KUKA KRL program: f1_Kuka_APT232T02S32.SRC

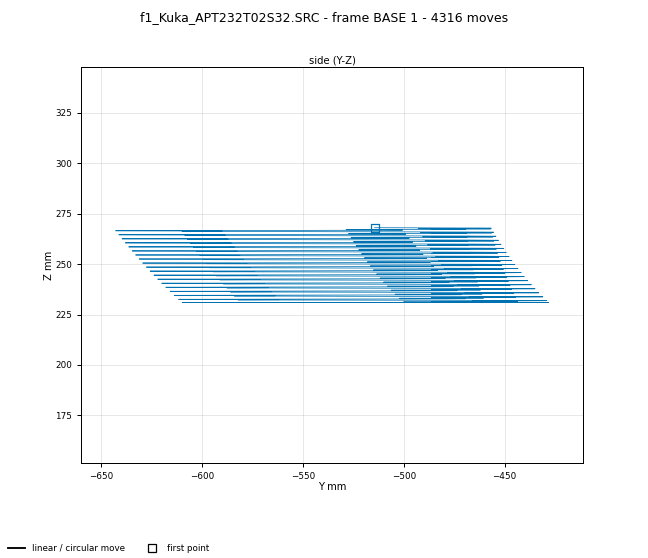
[picture p0: tool path of f1_Kuka_APT232T02S32.SRC in frame BASE 1, 4316 of 4317 moves have a stored position in this frame; points joined in program order, loops and branches not executed]
&ACCESS RVP
&REL 2
&PARAM TEMPLATE = C:\KRC\Roboter\Template\vorgabe
&PARAM EDITMASK = *
DEF f1_Kuka_APT232T02S32()


;FOLD INI;%{PE}%V3.2.0,%MKUKATPBASIS,%CINIT,%VCOMMON,%P
  ;FOLD BAS INI;%{E}%V3.2.0,%MKUKATPBASIS,%CINIT,%VINIT,%P
    GLOBAL INTERRUPT DECL 3 WHEN $STOPMESS==TRUE DO IR_STOPM ( )
    INTERRUPT ON 3
    BAS (#INITMOV,0 )
  ;ENDFOLD (BAS INI)
  ;FOLD USER INI;%{E}%V3.2.0,%MKUKATPUSER,%CINIT,%VINIT,%P
    ;Make your modifications here
  ;ENDFOLD (USER INI)
;ENDFOLD (INI)


;*** Make Null PTP Move
  PTP $pos_act

;*** Auto Load The Correct TOOL Data
  $tool=tool_data[2]

;*** Auto Load The Correct BASE Data
  $base=base_data[1]

  $ADVANCE = 5

;*** Restate Last Velocity
MMPM(30000.0)
SetRPM(8000)
LIN {X -0.230,Y -514.426,Z 267.989,A 0.000,B 0.000,C 90.000,E1 213.992} C_DIS
LIN {X 0.196,Y -508.743,Z 267.977,A 0.000,B 0.000,C 90.000,E1 211.878} C_DIS
LIN {X 0.196,Y -503.250,Z 267.966,A 0.000,B 0.000,C 90.000,E1 209.795} C_DIS
LIN {X -0.056,Y -498.886,Z 267.956,A 0.000,B 0.000,C 90.000,E1 208.025} C_DIS
LIN {X 0.152,Y -492.690,Z 267.941,A 0.000,B 0.000,C 90.000,E1 205.283} C_DIS
LIN {X 0.150,Y -488.290,Z 267.929,A 0.000,B 0.000,C 90.000,E1 203.153} C_DIS
LIN {X -0.154,Y -484.154,Z 267.917,A 0.000,B 0.000,C 90.000,E1 201.046} C_DIS
LIN {X 0.157,Y -479.821,Z 267.903,A 0.000,B 0.000,C 90.000,E1 198.544} C_DIS
LIN {X 0.025,Y -475.933,Z 267.889,A 0.000,B 0.000,C 90.000,E1 196.079} C_DIS
LIN {X 0.194,Y -471.593,Z 267.872,A 0.000,B 0.000,C 90.000,E1 192.939} C_DIS
LIN {X -0.221,Y -469.656,Z 267.863,A 0.000,B 0.000,C 90.000,E1 191.422} C_DIS
LIN {X 0.157,Y -466.683,Z 267.849,A 0.000,B 0.000,C 90.000,E1 188.859} C_DIS
LIN {X -0.167,Y -464.095,Z 267.835,A 0.000,B 0.000,C 90.000,E1 186.372} C_DIS
LIN {X 0.063,Y -462.670,Z 267.827,A 0.000,B 0.000,C 90.000,E1 184.759} C_DIS
LIN {X 0.115,Y -460.444,Z 267.811,A 0.000,B 0.000,C 90.000,E1 181.892} C_DIS
LIN {X 0.087,Y -458.680,Z 267.795,A 0.000,B 0.000,C 90.000,E1 179.026} C_DIS
LIN {X 0.013,Y -457.404,Z 267.779,A 0.000,B 0.000,C 90.000,E1 176.159} C_DIS
LIN {X 0.059,Y -456.833,Z 267.766,A 0.000,B 0.000,C 90.000,E1 173.913} C_DIS
LIN {X -0.071,Y -456.684,Z 267.756,A 0.000,B 0.000,C 90.000,E1 172.008} C_DIS
LIN {X -0.145,Y -456.659,Z 267.741,A 0.000,B 0.000,C 90.000,E1 169.454} C_DIS
LIN {X 0.170,Y -457.094,Z 267.729,A 0.000,B 0.000,C 90.000,E1 167.173} C_DIS
LIN {X 0.039,Y -457.494,Z 267.720,A 0.000,B 0.000,C 90.000,E1 165.589} C_DIS
LIN {X 0.182,Y -459.071,Z 267.700,A 0.000,B 0.000,C 90.000,E1 162.054} C_DIS
LIN {X -0.015,Y -461.188,Z 267.685,A 0.000,B 0.000,C 90.000,E1 159.209} C_DIS
LIN {X 0.063,Y -463.174,Z 267.672,A 0.000,B 0.000,C 90.000,E1 156.975} C_DIS
LIN {X -0.031,Y -466.661,Z 267.655,A 0.000,B 0.000,C 90.000,E1 153.819} C_DIS
LIN {X -0.099,Y -470.005,Z 267.641,A 0.000,B 0.000,C 90.000,E1 151.307} C_DIS
LIN {X 0.204,Y -473.267,Z 267.628,A 0.000,B 0.000,C 90.000,E1 149.076} C_DIS
LIN {X -0.166,Y -476.278,Z 267.618,A 0.000,B 0.000,C 90.000,E1 147.248} C_DIS
LIN {X -0.209,Y -479.468,Z 267.608,A 0.000,B 0.000,C 90.000,E1 145.388} C_DIS
LIN {X 0.091,Y -482.592,Z 267.597,A 0.000,B 0.000,C 90.000,E1 143.497} C_DIS
LIN {X -0.019,Y -485.558,Z 267.587,A 0.000,B 0.000,C 90.000,E1 141.662} C_DIS
LIN {X -0.030,Y -487.431,Z 267.580,A 0.000,B 0.000,C 90.000,E1 140.436} C_DIS
LIN {X -0.247,Y -489.510,Z 267.572,A 0.000,B 0.000,C 90.000,E1 138.933} C_DIS
LIN {X 0.062,Y -490.896,Z 267.565,A 0.000,B 0.000,C 90.000,E1 137.676} C_DIS
LIN {X -0.107,Y -491.742,Z 267.560,A 0.000,B 0.000,C 90.000,E1 136.782} C_DIS
LIN {X -0.293,Y -492.387,Z 267.555,A 0.000,B 0.000,C 90.000,E1 135.891} C_DIS
LIN {X 0.054,Y -492.760,Z 267.548,A 0.000,B 0.000,C 90.000,E1 134.636} C_DIS
LIN {X 0.233,Y -492.889,Z 267.543,A 0.000,B 0.000,C 90.000,E1 133.704} C_DIS
LIN {X -0.277,Y -492.766,Z 267.538,A 0.000,B 0.000,C 90.000,E1 132.852} C_DIS
LIN {X -0.090,Y -492.444,Z 267.533,A 0.000,B 0.000,C 90.000,E1 131.919} C_DIS
LIN {X -0.067,Y -491.559,Z 267.526,A 0.000,B 0.000,C 90.000,E1 130.701} C_DIS
LIN {X -0.061,Y -490.329,Z 267.519,A 0.000,B 0.000,C 90.000,E1 129.483} C_DIS
LIN {X -0.006,Y -488.945,Z 267.513,A 0.000,B 0.000,C 90.000,E1 128.257} C_DIS
LIN {X 0.033,Y -487.284,Z 267.506,A 0.000,B 0.000,C 90.000,E1 127.030} C_DIS
LIN {X 0.045,Y -485.471,Z 267.499,A 0.000,B 0.000,C 90.000,E1 125.804} C_DIS
LIN {X -0.039,Y -482.830,Z 267.490,A 0.000,B 0.000,C 90.000,E1 124.278} C_DIS
LIN {X -0.173,Y -480.059,Z 267.482,A 0.000,B 0.000,C 90.000,E1 122.752} C_DIS
LIN {X 0.034,Y -477.274,Z 267.473,A 0.000,B 0.000,C 90.000,E1 121.180} C_DIS
LIN {X 0.103,Y -474.436,Z 267.465,A 0.000,B 0.000,C 90.000,E1 119.617} C_DIS
LIN {X -0.166,Y -470.393,Z 267.453,A 0.000,B 0.000,C 90.000,E1 117.462} C_DIS
LIN {X 0.196,Y -467.495,Z 267.444,A 0.000,B 0.000,C 90.000,E1 115.848} C_DIS
LIN {X 0.156,Y -463.423,Z 267.432,A 0.000,B 0.000,C 90.000,E1 113.643} C_DIS
LIN {X 0.053,Y -461.128,Z 267.424,A 0.000,B 0.000,C 90.000,E1 112.386} C_DIS
LIN {X 0.164,Y -458.908,Z 267.417,A 0.000,B 0.000,C 90.000,E1 111.099} C_DIS
LIN {X -0.015,Y -456.909,Z 267.411,A 0.000,B 0.000,C 90.000,E1 109.939} C_DIS
LIN {X -0.055,Y -456.917,Z 267.411,A 0.000,B 0.000,C 90.000,E1 109.939} C_DIS
LIN {X 0.148,Y -457.785,Z 267.409,A 0.000,B 0.000,C 90.000,E1 109.504} C_DIS
LIN {X 0.113,Y -466.564,Z 267.386,A 0.000,B 0.000,C 90.000,E1 105.371} C_DIS
LIN {X 0.036,Y -467.351,Z 267.384,A 0.000,B 0.000,C 90.000,E1 105.064} C_DIS
LIN {X -0.160,Y -468.007,Z 267.382,A 0.000,B 0.000,C 90.000,E1 104.773} C_DIS
LIN {X -0.198,Y -476.222,Z 267.356,A 0.000,B 0.000,C 90.000,E1 100.074} C_DIS
LIN {X 0.056,Y -482.120,Z 267.330,A 0.000,B 0.000,C 90.000,E1 95.391} C_DIS
LIN {X -0.195,Y -485.524,Z 267.304,A 0.000,B 0.000,C 90.000,E1 90.802} C_DIS
LIN {X -0.161,Y -486.381,Z 267.281,A 0.000,B 0.000,C 90.000,E1 86.502} C_DIS
LIN {X 0.148,Y -486.354,Z 267.279,A 0.000,B 0.000,C 90.000,E1 86.159} C_DIS
LIN {X 0.227,Y -484.671,Z 267.253,A 0.000,B 0.000,C 90.000,E1 81.546} C_DIS
LIN {X 0.116,Y -480.589,Z 267.228,A 0.000,B 0.000,C 90.000,E1 76.937} C_DIS
LIN {X -0.172,Y -479.679,Z 267.224,A 0.000,B 0.000,C 90.000,E1 76.353} C_DIS
LIN {X -0.137,Y -474.020,Z 267.200,A 0.000,B 0.000,C 90.000,E1 72.000} C_DIS
LIN {X 0.177,Y -469.391,Z 267.186,A 0.000,B 0.000,C 90.000,E1 69.518} C_DIS
LIN {X 0.138,Y -469.387,Z 267.186,A 0.000,B 0.000,C 90.000,E1 69.518} C_DIS
LIN {X -0.086,Y -473.477,Z 267.177,A 0.000,B 0.000,C 90.000,E1 67.922} C_DIS
LIN {X -0.070,Y -478.382,Z 267.167,A 0.000,B 0.000,C 90.000,E1 66.049} C_DIS
LIN {X 0.060,Y -482.474,Z 267.158,A 0.000,B 0.000,C 90.000,E1 64.485} C_DIS
LIN {X -0.171,Y -487.487,Z 267.148,A 0.000,B 0.000,C 90.000,E1 62.666} C_DIS
LIN {X -0.098,Y -491.783,Z 267.140,A 0.000,B 0.000,C 90.000,E1 61.129} C_DIS
LIN {X 0.124,Y -496.998,Z 267.129,A 0.000,B 0.000,C 90.000,E1 59.282} C_DIS
LIN {X 0.139,Y -500.549,Z 267.123,A 0.000,B 0.000,C 90.000,E1 58.074} C_DIS
LIN {X -0.219,Y -504.000,Z 267.116,A 0.000,B 0.000,C 90.000,E1 56.914} C_DIS
LIN {X 0.173,Y -507.369,Z 267.109,A 0.000,B 0.000,C 90.000,E1 55.674} C_DIS
LIN {X 0.110,Y -511.278,Z 267.101,A 0.000,B 0.000,C 90.000,E1 54.196} C_DIS
LIN {X -0.219,Y -514.259,Z 267.095,A 0.000,B 0.000,C 90.000,E1 53.050} C_DIS
LIN {X 0.217,Y -516.997,Z 267.088,A 0.000,B 0.000,C 90.000,E1 51.823} C_DIS
LIN {X 0.231,Y -520.051,Z 267.080,A 0.000,B 0.000,C 90.000,E1 50.356} C_DIS
LIN {X -0.051,Y -522.220,Z 267.073,A 0.000,B 0.000,C 90.000,E1 49.218} C_DIS
LIN {X 0.137,Y -523.619,Z 267.069,A 0.000,B 0.000,C 90.000,E1 48.324} C_DIS
LIN {X -0.053,Y -524.883,Z 267.064,A 0.000,B 0.000,C 90.000,E1 47.472} C_DIS
LIN {X 0.081,Y -526.244,Z 267.057,A 0.000,B 0.000,C 90.000,E1 46.296} C_DIS
LIN {X -0.145,Y -527.243,Z 267.051,A 0.000,B 0.000,C 90.000,E1 45.162} C_DIS
LIN {X 0.068,Y -527.840,Z 267.046,A 0.000,B 0.000,C 90.000,E1 44.271} C_DIS
LIN {X -0.139,Y -528.298,Z 267.040,A 0.000,B 0.000,C 90.000,E1 43.137} C_DIS
LIN {X 0.039,Y -528.525,Z 267.033,A 0.000,B 0.000,C 90.000,E1 41.962} C_DIS
LIN {X 0.295,Y -528.546,Z 267.028,A 0.000,B 0.000,C 90.000,E1 41.067} C_DIS
LIN {X -0.189,Y -528.403,Z 267.024,A 0.000,B 0.000,C 90.000,E1 40.253} C_DIS
LIN {X 0.074,Y -528.098,Z 267.019,A 0.000,B 0.000,C 90.000,E1 39.358} C_DIS
LIN {X -0.137,Y -527.300,Z 267.011,A 0.000,B 0.000,C 90.000,E1 37.935} C_DIS
LIN {X -0.248,Y -526.425,Z 267.004,A 0.000,B 0.000,C 90.000,E1 36.790} C_DIS
LIN {X 0.057,Y -525.340,Z 266.998,A 0.000,B 0.000,C 90.000,E1 35.598} C_DIS
LIN {X 0.306,Y -523.688,Z 266.990,A 0.000,B 0.000,C 90.000,E1 34.119} C_DIS
LIN {X 0.273,Y -522.280,Z 266.983,A 0.000,B 0.000,C 90.000,E1 32.959} C_DIS
LIN {X -0.110,Y -520.461,Z 266.975,A 0.000,B 0.000,C 90.000,E1 31.544} C_DIS
LIN {X -0.154,Y -518.224,Z 266.965,A 0.000,B 0.000,C 90.000,E1 29.795} C_DIS
LIN {X -0.063,Y -516.128,Z 266.956,A 0.000,B 0.000,C 90.000,E1 28.025} C_DIS
LIN {X 0.197,Y -514.018,Z 266.946,A 0.000,B 0.000,C 90.000,E1 26.232} C_DIS
LIN {X -0.158,Y -511.788,Z 266.934,A 0.000,B 0.000,C 90.000,E1 24.207} C_DIS
LIN {X -0.058,Y -510.297,Z 266.926,A 0.000,B 0.000,C 90.000,E1 22.717} C_DIS
LIN {X 0.224,Y -508.272,Z 266.915,A 0.000,B 0.000,C 90.000,E1 20.610} C_DIS
LIN {X -0.004,Y -506.763,Z 266.905,A 0.000,B 0.000,C 90.000,E1 18.852} C_DIS
LIN {X 0.151,Y -505.095,Z 266.893,A 0.000,B 0.000,C 90.000,E1 16.749} C_DIS
LIN {X 0.183,Y -503.375,Z 266.880,A 0.000,B 0.000,C 90.000,E1 14.356} C_DIS
LIN {X 0.143,Y -501.822,Z 266.863,A 0.000,B 0.000,C 90.000,E1 11.366} C_DIS
LIN {X 0.017,Y -500.880,Z 266.848,A 0.000,B 0.000,C 90.000,E1 8.681} C_DIS
LIN {X -0.219,Y -500.607,Z 266.837,A 0.000,B 0.000,C 90.000,E1 6.606} C_DIS
LIN {X -0.176,Y -500.591,Z 266.822,A 0.000,B 0.000,C 90.000,E1 3.898} C_DIS
LIN {X -0.121,Y -501.117,Z 266.808,A 0.000,B 0.000,C 90.000,E1 1.489} C_DIS
LIN {X -0.044,Y -502.113,Z 266.796,A 0.000,B 0.000,C 90.000,E1 359.198} C_DIS
LIN {X 0.076,Y -503.746,Z 266.782,A 0.000,B 0.000,C 90.000,E1 356.788} C_DIS
LIN {X -0.150,Y -505.603,Z 266.771,A 0.000,B 0.000,C 90.000,E1 354.723} C_DIS
LIN {X -0.073,Y -507.065,Z 266.762,A 0.000,B 0.000,C 90.000,E1 353.223} C_DIS
LIN {X 0.174,Y -512.463,Z 266.743,A 0.000,B 0.000,C 90.000,E1 349.634} C_DIS
LIN {X 0.075,Y -519.137,Z 266.726,A 0.000,B 0.000,C 90.000,E1 346.700} C_DIS
LIN {X 0.181,Y -523.006,Z 266.718,A 0.000,B 0.000,C 90.000,E1 345.227} C_DIS
LIN {X -0.168,Y -526.106,Z 266.712,A 0.000,B 0.000,C 90.000,E1 344.102} C_DIS
LIN {X 0.250,Y -533.219,Z 266.697,A 0.000,B 0.000,C 90.000,E1 341.456} C_DIS
LIN {X 0.138,Y -539.356,Z 266.686,A 0.000,B 0.000,C 90.000,E1 339.464} C_DIS
LIN {X -0.207,Y -546.932,Z 266.673,A 0.000,B 0.000,C 90.000,E1 337.230} C_DIS
LIN {X 0.081,Y -551.791,Z 266.666,A 0.000,B 0.000,C 90.000,E1 335.793} C_DIS
LIN {X -0.049,Y -556.779,Z 266.658,A 0.000,B 0.000,C 90.000,E1 334.409} C_DIS
LIN {X -0.247,Y -563.958,Z 266.647,A 0.000,B 0.000,C 90.000,E1 332.487} C_DIS
LIN {X -0.243,Y -568.105,Z 266.641,A 0.000,B 0.000,C 90.000,E1 331.385} C_DIS
LIN {X -0.073,Y -573.033,Z 266.633,A 0.000,B 0.000,C 90.000,E1 329.999} C_DIS
LIN {X 0.184,Y -577.781,Z 266.626,A 0.000,B 0.000,C 90.000,E1 328.614} C_DIS
LIN {X -0.132,Y -584.424,Z 266.615,A 0.000,B 0.000,C 90.000,E1 326.755} C_DIS
LIN {X 0.003,Y -590.503,Z 266.606,A 0.000,B 0.000,C 90.000,E1 325.135} C_DIS
LIN {X -0.029,Y -596.487,Z 266.598,A 0.000,B 0.000,C 90.000,E1 323.543} C_DIS
LIN {X 0.069,Y -600.158,Z 266.592,A 0.000,B 0.000,C 90.000,E1 322.477} C_DIS
LIN {X -0.010,Y -604.543,Z 266.584,A 0.000,B 0.000,C 90.000,E1 321.170} C_DIS
LIN {X 0.368,Y -608.852,Z 266.577,A 0.000,B 0.000,C 90.000,E1 319.828} C_DIS
LIN {X -0.222,Y -613.909,Z 266.568,A 0.000,B 0.000,C 90.000,E1 318.324} C_DIS
LIN {X 0.267,Y -618.187,Z 266.561,A 0.000,B 0.000,C 90.000,E1 316.986} C_DIS
LIN {X 0.254,Y -620.662,Z 266.557,A 0.000,B 0.000,C 90.000,E1 316.215} C_DIS
LIN {X -0.026,Y -624.392,Z 266.550,A 0.000,B 0.000,C 90.000,E1 314.960} C_DIS
LIN {X -0.116,Y -627.253,Z 266.544,A 0.000,B 0.000,C 90.000,E1 313.947} C_DIS
LIN {X -0.161,Y -629.986,Z 266.538,A 0.000,B 0.000,C 90.000,E1 312.933} C_DIS
LIN {X -0.167,Y -632.434,Z 266.533,A 0.000,B 0.000,C 90.000,E1 311.919} C_DIS
LIN {X -0.147,Y -634.695,Z 266.527,A 0.000,B 0.000,C 90.000,E1 310.906} C_DIS
LIN {X -0.029,Y -636.679,Z 266.522,A 0.000,B 0.000,C 90.000,E1 309.886} C_DIS
LIN {X -0.370,Y -638.383,Z 266.516,A 0.000,B 0.000,C 90.000,E1 308.910} C_DIS
LIN {X 0.206,Y -640.180,Z 266.509,A 0.000,B 0.000,C 90.000,E1 307.604} C_DIS
LIN {X 0.406,Y -641.435,Z 266.503,A 0.000,B 0.000,C 90.000,E1 306.583} C_DIS
LIN {X -0.172,Y -642.058,Z 266.499,A 0.000,B 0.000,C 90.000,E1 305.884} C_DIS
LIN {X 0.157,Y -642.446,Z 266.495,A 0.000,B 0.000,C 90.000,E1 305.105} C_DIS
LIN {X -0.409,Y -642.645,Z 266.491,A 0.000,B 0.000,C 90.000,E1 304.405} C_DIS
LIN {X 0.370,Y -642.696,Z 266.484,A 0.000,B 0.000,C 90.000,E1 303.086} C_DIS
LIN {X 0.339,Y -642.403,Z 266.480,A 0.000,B 0.000,C 90.000,E1 302.339} C_DIS
LIN {X 0.305,Y -641.761,Z 266.476,A 0.000,B 0.000,C 90.000,E1 301.592} C_DIS
LIN {X -0.126,Y -641.196,Z 266.473,A 0.000,B 0.000,C 90.000,E1 301.131} C_DIS
LIN {X -0.175,Y -639.987,Z 266.469,A 0.000,B 0.000,C 90.000,E1 300.384} C_DIS
LIN {X 0.364,Y -638.024,Z 266.463,A 0.000,B 0.000,C 90.000,E1 299.333} C_DIS
LIN {X 0.061,Y -635.155,Z 266.456,A 0.000,B 0.000,C 90.000,E1 298.103} C_DIS
LIN {X -0.324,Y -632.632,Z 266.451,A 0.000,B 0.000,C 90.000,E1 297.129} C_DIS
LIN {X -0.150,Y -629.298,Z 266.444,A 0.000,B 0.000,C 90.000,E1 295.848} C_DIS
LIN {X -0.273,Y -624.517,Z 266.434,A 0.000,B 0.000,C 90.000,E1 294.079} C_DIS
LIN {X 0.067,Y -621.195,Z 266.427,A 0.000,B 0.000,C 90.000,E1 292.770} C_DIS
LIN {X -0.178,Y -615.973,Z 266.415,A 0.000,B 0.000,C 90.000,E1 290.737} C_DIS
LIN {X 0.059,Y -611.666,Z 266.405,A 0.000,B 0.000,C 90.000,E1 288.906} C_DIS
LIN {X -0.044,Y -605.942,Z 266.391,A 0.000,B 0.000,C 90.000,E1 286.315} C_DIS
LIN {X -0.282,Y -601.908,Z 266.379,A 0.000,B 0.000,C 90.000,E1 284.245} C_DIS
LIN {X 0.146,Y -596.652,Z 266.360,A 0.000,B 0.000,C 90.000,E1 280.782} C_DIS
LIN {X -0.261,Y -593.058,Z 266.342,A 0.000,B 0.000,C 90.000,E1 277.644} C_DIS
LIN {X -0.064,Y -590.974,Z 266.326,A 0.000,B 0.000,C 90.000,E1 274.702} C_DIS
LIN {X 0.269,Y -589.995,Z 266.311,A 0.000,B 0.000,C 90.000,E1 272.007} C_DIS
LIN {X 0.003,Y -590.230,Z 266.292,A 0.000,B 0.000,C 90.000,E1 268.568} C_DIS
LIN {X -0.149,Y -592.176,Z 266.273,A 0.000,B 0.000,C 90.000,E1 265.122} C_DIS
LIN {X -0.173,Y -594.805,Z 266.258,A 0.000,B 0.000,C 90.000,E1 262.470} C_DIS
LIN {X -0.052,Y -599.032,Z 266.241,A 0.000,B 0.000,C 90.000,E1 259.285} C_DIS
LIN {X -0.005,Y -601.486,Z 266.232,A 0.000,B 0.000,C 90.000,E1 257.701} C_DIS
LIN {X 0.097,Y -604.047,Z 266.223,A 0.000,B 0.000,C 90.000,E1 256.117} C_DIS
LIN {X -0.192,Y -606.411,Z 266.214,A 0.000,B 0.000,C 90.000,E1 254.574} C_DIS
LIN {X -0.235,Y -607.542,Z 266.210,A 0.000,B 0.000,C 90.000,E1 253.795} C_DIS
LIN {X 0.319,Y -608.398,Z 266.206,A 0.000,B 0.000,C 90.000,E1 252.960} C_DIS
LIN {X 0.298,Y -608.926,Z 266.201,A 0.000,B 0.000,C 90.000,E1 252.181} C_DIS
LIN {X -0.050,Y -609.582,Z 266.194,A 0.000,B 0.000,C 90.000,E1 250.913} C_DIS
LIN {X -0.128,Y -609.794,Z 266.188,A 0.000,B 0.000,C 90.000,E1 249.880} C_DIS
LIN {X 0.064,Y -609.722,Z 266.184,A 0.000,B 0.000,C 90.000,E1 249.082} C_DIS
LIN {X 0.256,Y -609.357,Z 266.180,A 0.000,B 0.000,C 90.000,E1 248.284} C_DIS
LIN {X -0.122,Y -608.730,Z 266.175,A 0.000,B 0.000,C 90.000,E1 247.539} C_DIS
LIN {X 0.055,Y -607.911,Z 266.171,A 0.000,B 0.000,C 90.000,E1 246.741} C_DIS
LIN {X -0.094,Y -606.864,Z 266.167,A 0.000,B 0.000,C 90.000,E1 245.973} C_DIS
LIN {X -0.003,Y -605.009,Z 266.161,A 0.000,B 0.000,C 90.000,E1 244.921} C_DIS
LIN {X -0.173,Y -603.330,Z 266.156,A 0.000,B 0.000,C 90.000,E1 244.152} C_DIS
LIN {X 0.045,Y -600.272,Z 266.149,A 0.000,B 0.000,C 90.000,E1 242.820} C_DIS
LIN {X 0.029,Y -597.617,Z 266.143,A 0.000,B 0.000,C 90.000,E1 241.769} C_DIS
LIN {X -0.200,Y -593.379,Z 266.134,A 0.000,B 0.000,C 90.000,E1 240.205} C_DIS
LIN {X -0.006,Y -590.340,Z 266.129,A 0.000,B 0.000,C 90.000,E1 239.125} C_DIS
LIN {X -0.158,Y -587.134,Z 266.123,A 0.000,B 0.000,C 90.000,E1 238.074} C_DIS
LIN {X 0.125,Y -582.839,Z 266.115,A 0.000,B 0.000,C 90.000,E1 236.707} C_DIS
LIN {X 0.175,Y -576.795,Z 266.105,A 0.000,B 0.000,C 90.000,E1 234.815} C_DIS
LIN {X -0.060,Y -571.748,Z 266.096,A 0.000,B 0.000,C 90.000,E1 233.210} C_DIS
LIN {X 0.154,Y -567.561,Z 266.088,A 0.000,B 0.000,C 90.000,E1 231.823} C_DIS
LIN {X 0.067,Y -561.705,Z 266.077,A 0.000,B 0.000,C 90.000,E1 229.908} C_DIS
LIN {X 0.112,Y -556.554,Z 266.068,A 0.000,B 0.000,C 90.000,E1 228.243} C_DIS
LIN {X -0.015,Y -552.185,Z 266.060,A 0.000,B 0.000,C 90.000,E1 226.863} C_DIS
LIN {X 0.168,Y -546.868,Z 266.051,A 0.000,B 0.000,C 90.000,E1 225.162} C_DIS
LIN {X -0.148,Y -542.407,Z 266.043,A 0.000,B 0.000,C 90.000,E1 223.785} C_DIS
LIN {X -0.150,Y -537.062,Z 266.034,A 0.000,B 0.000,C 90.000,E1 222.081} C_DIS
LIN {X 0.153,Y -533.552,Z 266.027,A 0.000,B 0.000,C 90.000,E1 220.906} C_DIS
LIN {X -0.012,Y -527.392,Z 266.016,A 0.000,B 0.000,C 90.000,E1 218.910} C_DIS
LIN {X 0.163,Y -523.022,Z 266.008,A 0.000,B 0.000,C 90.000,E1 217.443} C_DIS
LIN {X -0.061,Y -518.815,Z 266.000,A 0.000,B 0.000,C 90.000,E1 216.011} C_DIS
LIN {X 0.332,Y -512.957,Z 265.989,A 0.000,B 0.000,C 90.000,E1 213.913} C_DIS
LIN {X 0.009,Y -507.262,Z 265.977,A 0.000,B 0.000,C 90.000,E1 211.878} C_DIS
LIN {X 0.027,Y -501.052,Z 265.964,A 0.000,B 0.000,C 90.000,E1 209.489} C_DIS
LIN {X 0.015,Y -495.970,Z 265.952,A 0.000,B 0.000,C 90.000,E1 207.385} C_DIS
LIN {X -0.148,Y -491.227,Z 265.940,A 0.000,B 0.000,C 90.000,E1 205.283} C_DIS
LIN {X 0.025,Y -486.245,Z 265.927,A 0.000,B 0.000,C 90.000,E1 202.823} C_DIS
LIN {X -0.061,Y -481.608,Z 265.913,A 0.000,B 0.000,C 90.000,E1 200.375} C_DIS
LIN {X 0.185,Y -477.914,Z 265.901,A 0.000,B 0.000,C 90.000,E1 198.181} C_DIS
LIN {X 0.032,Y -474.562,Z 265.889,A 0.000,B 0.000,C 90.000,E1 196.024} C_DIS
LIN {X -0.124,Y -470.656,Z 265.873,A 0.000,B 0.000,C 90.000,E1 193.231} C_DIS
LIN {X -0.099,Y -468.718,Z 265.865,A 0.000,B 0.000,C 90.000,E1 191.658} C_DIS
LIN {X -0.207,Y -465.737,Z 265.851,A 0.000,B 0.000,C 90.000,E1 189.151} C_DIS
LIN {X -0.090,Y -463.098,Z 265.837,A 0.000,B 0.000,C 90.000,E1 186.606} C_DIS
LIN {X 0.128,Y -461.672,Z 265.828,A 0.000,B 0.000,C 90.000,E1 184.992} C_DIS
LIN {X -0.021,Y -459.613,Z 265.814,A 0.000,B 0.000,C 90.000,E1 182.465} C_DIS
LIN {X -0.008,Y -458.131,Z 265.801,A 0.000,B 0.000,C 90.000,E1 180.229} C_DIS
LIN {X -0.232,Y -457.055,Z 265.791,A 0.000,B 0.000,C 90.000,E1 178.339} C_DIS
LIN {X 0.182,Y -456.161,Z 265.778,A 0.000,B 0.000,C 90.000,E1 176.045} C_DIS
LIN {X 0.192,Y -455.610,Z 265.766,A 0.000,B 0.000,C 90.000,E1 173.799} C_DIS
LIN {X 0.031,Y -455.469,Z 265.755,A 0.000,B 0.000,C 90.000,E1 171.894} C_DIS
LIN {X 0.144,Y -455.497,Z 265.743,A 0.000,B 0.000,C 90.000,E1 169.634} C_DIS
LIN {X 0.190,Y -456.013,Z 265.728,A 0.000,B 0.000,C 90.000,E1 167.061} C_DIS
LIN {X -0.082,Y -456.533,Z 265.718,A 0.000,B 0.000,C 90.000,E1 165.172} C_DIS
LIN {X -0.223,Y -457.868,Z 265.702,A 0.000,B 0.000,C 90.000,E1 162.308} C_DIS
LIN {X 0.201,Y -459.677,Z 265.687,A 0.000,B 0.000,C 90.000,E1 159.699} C_DIS
LIN {X -0.015,Y -461.941,Z 265.673,A 0.000,B 0.000,C 90.000,E1 157.177} C_DIS
LIN {X -0.173,Y -465.397,Z 265.656,A 0.000,B 0.000,C 90.000,E1 154.024} C_DIS
LIN {X -0.135,Y -469.145,Z 265.640,A 0.000,B 0.000,C 90.000,E1 151.179} C_DIS
LIN {X -0.089,Y -472.944,Z 265.626,A 0.000,B 0.000,C 90.000,E1 148.663} C_DIS
LIN {X -0.281,Y -476.473,Z 265.614,A 0.000,B 0.000,C 90.000,E1 146.501} C_DIS
LIN {X -0.045,Y -478.628,Z 265.607,A 0.000,B 0.000,C 90.000,E1 145.229} C_DIS
LIN {X -0.239,Y -481.210,Z 265.598,A 0.000,B 0.000,C 90.000,E1 143.703} C_DIS
LIN {X 0.069,Y -483.197,Z 265.591,A 0.000,B 0.000,C 90.000,E1 142.431} C_DIS
LIN {X -0.056,Y -485.131,Z 265.585,A 0.000,B 0.000,C 90.000,E1 141.215} C_DIS
LIN {X -0.074,Y -486.918,Z 265.578,A 0.000,B 0.000,C 90.000,E1 139.989} C_DIS
LIN {X -0.131,Y -488.543,Z 265.571,A 0.000,B 0.000,C 90.000,E1 138.771} C_DIS
LIN {X -0.165,Y -489.894,Z 265.564,A 0.000,B 0.000,C 90.000,E1 137.553} C_DIS
LIN {X 0.150,Y -490.929,Z 265.557,A 0.000,B 0.000,C 90.000,E1 136.296} C_DIS
LIN {X -0.041,Y -491.380,Z 265.552,A 0.000,B 0.000,C 90.000,E1 135.405} C_DIS
LIN {X -0.227,Y -491.642,Z 265.547,A 0.000,B 0.000,C 90.000,E1 134.514} C_DIS
LIN {X 0.118,Y -491.730,Z 265.540,A 0.000,B 0.000,C 90.000,E1 133.257} C_DIS
LIN {X 0.097,Y -491.394,Z 265.534,A 0.000,B 0.000,C 90.000,E1 132.043} C_DIS
LIN {X -0.062,Y -490.847,Z 265.529,A 0.000,B 0.000,C 90.000,E1 131.148} C_DIS
LIN {X -0.221,Y -490.055,Z 265.524,A 0.000,B 0.000,C 90.000,E1 130.253} C_DIS
LIN {X -0.022,Y -488.410,Z 265.515,A 0.000,B 0.000,C 90.000,E1 128.705} C_DIS
LIN {X -0.208,Y -487.302,Z 265.510,A 0.000,B 0.000,C 90.000,E1 127.810} C_DIS
LIN {X -0.196,Y -485.597,Z 265.503,A 0.000,B 0.000,C 90.000,E1 126.583} C_DIS
LIN {X 0.179,Y -483.700,Z 265.496,A 0.000,B 0.000,C 90.000,E1 125.311} C_DIS
LIN {X 0.061,Y -481.021,Z 265.488,A 0.000,B 0.000,C 90.000,E1 123.785} C_DIS
LIN {X 0.089,Y -478.811,Z 265.481,A 0.000,B 0.000,C 90.000,E1 122.546} C_DIS
LIN {X -0.174,Y -476.612,Z 265.474,A 0.000,B 0.000,C 90.000,E1 121.337} C_DIS
LIN {X -0.102,Y -473.191,Z 265.464,A 0.000,B 0.000,C 90.000,E1 119.461} C_DIS
LIN {X 0.001,Y -469.179,Z 265.451,A 0.000,B 0.000,C 90.000,E1 117.257} C_DIS
LIN {X 0.130,Y -466.273,Z 265.443,A 0.000,B 0.000,C 90.000,E1 115.668} C_DIS
LIN {X 0.063,Y -462.238,Z 265.430,A 0.000,B 0.000,C 90.000,E1 113.462} C_DIS
LIN {X -0.217,Y -458.851,Z 265.420,A 0.000,B 0.000,C 90.000,E1 111.589} C_DIS
LIN {X -0.010,Y -456.401,Z 265.412,A 0.000,B 0.000,C 90.000,E1 110.120} C_DIS
LIN {X -0.050,Y -456.402,Z 265.412,A 0.000,B 0.000,C 90.000,E1 110.120} C_DIS
LIN {X 0.103,Y -457.569,Z 265.409,A 0.000,B 0.000,C 90.000,E1 109.631} C_DIS
LIN {X 0.189,Y -466.270,Z 265.386,A 0.000,B 0.000,C 90.000,E1 105.481} C_DIS
LIN {X -0.208,Y -467.823,Z 265.383,A 0.000,B 0.000,C 90.000,E1 104.898} C_DIS
LIN {X -0.238,Y -476.030,Z 265.357,A 0.000,B 0.000,C 90.000,E1 100.197} C_DIS
LIN {X 0.067,Y -477.355,Z 265.350,A 0.000,B 0.000,C 90.000,E1 98.916} C_DIS
LIN {X 0.036,Y -481.962,Z 265.331,A 0.000,B 0.000,C 90.000,E1 95.511} C_DIS
LIN {X 0.170,Y -482.350,Z 265.327,A 0.000,B 0.000,C 90.000,E1 94.878} C_DIS
LIN {X -0.178,Y -485.422,Z 265.305,A 0.000,B 0.000,C 90.000,E1 90.917} C_DIS
LIN {X -0.041,Y -485.506,Z 265.302,A 0.000,B 0.000,C 90.000,E1 90.286} C_DIS
LIN {X -0.146,Y -486.372,Z 265.281,A 0.000,B 0.000,C 90.000,E1 86.617} C_DIS
LIN {X 0.165,Y -486.367,Z 265.279,A 0.000,B 0.000,C 90.000,E1 86.274} C_DIS
LIN {X -0.007,Y -485.229,Z 265.268,A 0.000,B 0.000,C 90.000,E1 84.147} C_DIS
LIN {X 0.253,Y -484.691,Z 265.254,A 0.000,B 0.000,C 90.000,E1 81.659} C_DIS
LIN {X 0.050,Y -484.469,Z 265.252,A 0.000,B 0.000,C 90.000,E1 81.376} C_DIS
LIN {X 0.054,Y -480.654,Z 265.228,A 0.000,B 0.000,C 90.000,E1 77.061} C_DIS
LIN {X 0.020,Y -480.389,Z 265.227,A 0.000,B 0.000,C 90.000,E1 76.756} C_DIS
LIN {X -0.206,Y -474.179,Z 265.201,A 0.000,B 0.000,C 90.000,E1 72.127} C_DIS
LIN {X -0.049,Y -471.762,Z 265.194,A 0.000,B 0.000,C 90.000,E1 70.859} C_DIS
LIN {X -0.057,Y -469.037,Z 265.185,A 0.000,B 0.000,C 90.000,E1 69.337} C_DIS
LIN {X -0.097,Y -469.049,Z 265.185,A 0.000,B 0.000,C 90.000,E1 69.337} C_DIS
LIN {X -0.066,Y -473.908,Z 265.174,A 0.000,B 0.000,C 90.000,E1 67.411} C_DIS
LIN {X -0.012,Y -477.998,Z 265.166,A 0.000,B 0.000,C 90.000,E1 65.845} C_DIS
LIN {X 0.127,Y -481.291,Z 265.159,A 0.000,B 0.000,C 90.000,E1 64.588} C_DIS
LIN {X 0.093,Y -487.131,Z 265.147,A 0.000,B 0.000,C 90.000,E1 62.436} C_DIS
LIN {X -0.044,Y -491.401,Z 265.138,A 0.000,B 0.000,C 90.000,E1 60.923} C_DIS
LIN {X 0.023,Y -497.530,Z 265.127,A 0.000,B 0.000,C 90.000,E1 58.791} C_DIS
LIN {X -0.078,Y -501.919,Z 265.118,A 0.000,B 0.000,C 90.000,E1 57.296} C_DIS
LIN {X -0.103,Y -506.109,Z 265.110,A 0.000,B 0.000,C 90.000,E1 55.801} C_DIS
LIN {X 0.227,Y -510.027,Z 265.102,A 0.000,B 0.000,C 90.000,E1 54.276} C_DIS
LIN {X -0.203,Y -513.692,Z 265.094,A 0.000,B 0.000,C 90.000,E1 52.844} C_DIS
LIN {X 0.222,Y -516.407,Z 265.087,A 0.000,B 0.000,C 90.000,E1 51.618} C_DIS
LIN {X -0.178,Y -519.391,Z 265.079,A 0.000,B 0.000,C 90.000,E1 50.194} C_DIS
LIN {X -0.077,Y -521.495,Z 265.072,A 0.000,B 0.000,C 90.000,E1 49.013} C_DIS
LIN {X 0.005,Y -523.254,Z 265.066,A 0.000,B 0.000,C 90.000,E1 47.838} C_DIS
LIN {X 0.120,Y -524.724,Z 265.059,A 0.000,B 0.000,C 90.000,E1 46.662} C_DIS
LIN {X -0.059,Y -525.534,Z 265.055,A 0.000,B 0.000,C 90.000,E1 45.810} C_DIS
LIN {X -0.177,Y -526.041,Z 265.051,A 0.000,B 0.000,C 90.000,E1 45.243} C_DIS
LIN {X 0.023,Y -526.619,Z 265.046,A 0.000,B 0.000,C 90.000,E1 44.352} C_DIS
LIN {X 0.182,Y -527.078,Z 265.040,A 0.000,B 0.000,C 90.000,E1 43.176} C_DIS
LIN {X -0.041,Y -527.297,Z 265.034,A 0.000,B 0.000,C 90.000,E1 42.043} C_DIS
LIN {X 0.200,Y -527.326,Z 265.029,A 0.000,B 0.000,C 90.000,E1 41.148} C_DIS
LIN {X 0.047,Y -527.195,Z 265.024,A 0.000,B 0.000,C 90.000,E1 40.297} C_DIS
LIN {X -0.045,Y -526.871,Z 265.019,A 0.000,B 0.000,C 90.000,E1 39.439} C_DIS
LIN {X 0.141,Y -526.066,Z 265.011,A 0.000,B 0.000,C 90.000,E1 37.971} C_DIS
LIN {X 0.020,Y -525.190,Z 265.005,A 0.000,B 0.000,C 90.000,E1 36.824} C_DIS
LIN {X -0.113,Y -524.086,Z 264.998,A 0.000,B 0.000,C 90.000,E1 35.678} C_DIS
LIN {X 0.116,Y -522.384,Z 264.990,A 0.000,B 0.000,C 90.000,E1 34.199} C_DIS
LIN {X 0.069,Y -520.955,Z 264.984,A 0.000,B 0.000,C 90.000,E1 33.038} C_DIS
LIN {X 0.314,Y -518.685,Z 264.974,A 0.000,B 0.000,C 90.000,E1 31.258} C_DIS
LIN {X 0.328,Y -516.083,Z 264.962,A 0.000,B 0.000,C 90.000,E1 29.205} C_DIS
LIN {X 0.019,Y -514.330,Z 264.954,A 0.000,B 0.000,C 90.000,E1 27.769} C_DIS
LIN {X 0.240,Y -512.209,Z 264.945,A 0.000,B 0.000,C 90.000,E1 25.976} C_DIS
LIN {X -0.056,Y -509.702,Z 264.931,A 0.000,B 0.000,C 90.000,E1 23.643} C_DIS
LIN {X 0.107,Y -507.876,Z 264.921,A 0.000,B 0.000,C 90.000,E1 21.844} C_DIS
LIN {X 0.231,Y -505.727,Z 264.908,A 0.000,B 0.000,C 90.000,E1 19.450} C_DIS
LIN {X -0.138,Y -504.489,Z 264.900,A 0.000,B 0.000,C 90.000,E1 18.000} C_DIS
LIN {X -0.121,Y -503.092,Z 264.890,A 0.000,B 0.000,C 90.000,E1 16.205} C_DIS
LIN {X 0.204,Y -501.435,Z 264.877,A 0.000,B 0.000,C 90.000,E1 13.772} C_DIS
LIN {X -0.246,Y -500.219,Z 264.863,A 0.000,B 0.000,C 90.000,E1 11.422} C_DIS
LIN {X 0.065,Y -499.269,Z 264.848,A 0.000,B 0.000,C 90.000,E1 8.681} C_DIS
LIN {X -0.212,Y -498.960,Z 264.837,A 0.000,B 0.000,C 90.000,E1 6.606} C_DIS
LIN {X -0.224,Y -498.940,Z 264.822,A 0.000,B 0.000,C 90.000,E1 3.898} C_DIS
LIN {X 0.154,Y -499.539,Z 264.807,A 0.000,B 0.000,C 90.000,E1 1.146} C_DIS
LIN {X -0.179,Y -500.594,Z 264.794,A 0.000,B 0.000,C 90.000,E1 358.912} C_DIS
LIN {X -0.230,Y -502.521,Z 264.779,A 0.000,B 0.000,C 90.000,E1 356.216} C_DIS
LIN {X 0.046,Y -504.416,Z 264.767,A 0.000,B 0.000,C 90.000,E1 354.090} C_DIS
LIN {X 0.210,Y -508.638,Z 264.749,A 0.000,B 0.000,C 90.000,E1 350.792} C_DIS
LIN {X -0.155,Y -512.525,Z 264.737,A 0.000,B 0.000,C 90.000,E1 348.757} C_DIS
LIN {X -0.134,Y -520.626,Z 264.720,A 0.000,B 0.000,C 90.000,E1 345.519} C_DIS
LIN {X 0.134,Y -524.485,Z 264.711,A 0.000,B 0.000,C 90.000,E1 344.031} C_DIS
LIN {X -0.155,Y -531.647,Z 264.697,A 0.000,B 0.000,C 90.000,E1 341.456} C_DIS
LIN {X 0.120,Y -539.675,Z 264.683,A 0.000,B 0.000,C 90.000,E1 338.847} C_DIS
LIN {X -0.203,Y -545.425,Z 264.673,A 0.000,B 0.000,C 90.000,E1 337.177} C_DIS
LIN {X -0.208,Y -549.305,Z 264.667,A 0.000,B 0.000,C 90.000,E1 336.049} C_DIS
LIN {X -0.092,Y -556.276,Z 264.656,A 0.000,B 0.000,C 90.000,E1 334.076} C_DIS
LIN {X -0.096,Y -562.467,Z 264.647,A 0.000,B 0.000,C 90.000,E1 332.410} C_DIS
LIN {X -0.107,Y -566.631,Z 264.641,A 0.000,B 0.000,C 90.000,E1 331.307} C_DIS
LIN {X 0.043,Y -571.611,Z 264.633,A 0.000,B 0.000,C 90.000,E1 329.921} C_DIS
LIN {X 0.280,Y -576.381,Z 264.625,A 0.000,B 0.000,C 90.000,E1 328.535} C_DIS
LIN {X -0.035,Y -585.059,Z 264.612,A 0.000,B 0.000,C 90.000,E1 326.135} C_DIS
LIN {X 0.246,Y -590.165,Z 264.604,A 0.000,B 0.000,C 90.000,E1 324.769} C_DIS
LIN {X 0.254,Y -594.199,Z 264.599,A 0.000,B 0.000,C 90.000,E1 323.703} C_DIS
LIN {X -0.159,Y -597.899,Z 264.593,A 0.000,B 0.000,C 90.000,E1 322.683} C_DIS
LIN {X -0.048,Y -601.417,Z 264.587,A 0.000,B 0.000,C 90.000,E1 321.618} C_DIS
LIN {X 0.272,Y -605.782,Z 264.579,A 0.000,B 0.000,C 90.000,E1 320.275} C_DIS
LIN {X -0.187,Y -610.054,Z 264.572,A 0.000,B 0.000,C 90.000,E1 319.013} C_DIS
LIN {X -0.355,Y -615.227,Z 264.564,A 0.000,B 0.000,C 90.000,E1 317.472} C_DIS
LIN {X 0.312,Y -618.646,Z 264.558,A 0.000,B 0.000,C 90.000,E1 316.377} C_DIS
LIN {X -0.295,Y -621.770,Z 264.552,A 0.000,B 0.000,C 90.000,E1 315.405} C_DIS
LIN {X 0.021,Y -624.706,Z 264.546,A 0.000,B 0.000,C 90.000,E1 314.352} C_DIS
LIN {X -0.184,Y -628.148,Z 264.539,A 0.000,B 0.000,C 90.000,E1 313.095} C_DIS
LIN {X -0.092,Y -630.075,Z 264.535,A 0.000,B 0.000,C 90.000,E1 312.324} C_DIS
LIN {X 0.019,Y -631.823,Z 264.531,A 0.000,B 0.000,C 90.000,E1 311.553} C_DIS
LIN {X 0.033,Y -633.923,Z 264.525,A 0.000,B 0.000,C 90.000,E1 310.539} C_DIS
LIN {X -0.231,Y -635.364,Z 264.521,A 0.000,B 0.000,C 90.000,E1 309.806} C_DIS
LIN {X 0.305,Y -637.044,Z 264.515,A 0.000,B 0.000,C 90.000,E1 308.749} C_DIS
LIN {X -0.042,Y -638.803,Z 264.508,A 0.000,B 0.000,C 90.000,E1 307.523} C_DIS
LIN {X -0.262,Y -639.719,Z 264.504,A 0.000,B 0.000,C 90.000,E1 306.790} C_DIS
LIN {X 0.038,Y -640.392,Z 264.500,A 0.000,B 0.000,C 90.000,E1 306.011} C_DIS
LIN {X 0.346,Y -640.799,Z 264.496,A 0.000,B 0.000,C 90.000,E1 305.231} C_DIS
LIN {X -0.198,Y -641.052,Z 264.490,A 0.000,B 0.000,C 90.000,E1 304.278} C_DIS
LIN {X 0.158,Y -641.111,Z 264.485,A 0.000,B 0.000,C 90.000,E1 303.245} C_DIS
LIN {X 0.117,Y -640.865,Z 264.481,A 0.000,B 0.000,C 90.000,E1 302.498} C_DIS
LIN {X 0.020,Y -640.539,Z 264.478,A 0.000,B 0.000,C 90.000,E1 302.005} C_DIS
LIN {X -0.031,Y -639.728,Z 264.474,A 0.000,B 0.000,C 90.000,E1 301.258} C_DIS
LIN {X -0.096,Y -638.605,Z 264.470,A 0.000,B 0.000,C 90.000,E1 300.512} C_DIS
LIN {X 0.108,Y -636.685,Z 264.464,A 0.000,B 0.000,C 90.000,E1 299.489} C_DIS
LIN {X 0.052,Y -634.455,Z 264.458,A 0.000,B 0.000,C 90.000,E1 298.487} C_DIS
LIN {X -0.307,Y -631.384,Z 264.451,A 0.000,B 0.000,C 90.000,E1 297.257} C_DIS
LIN {X -0.153,Y -628.040,Z 264.444,A 0.000,B 0.000,C 90.000,E1 295.976} C_DIS
LIN {X -0.306,Y -623.238,Z 264.434,A 0.000,B 0.000,C 90.000,E1 294.207} C_DIS
LIN {X 0.005,Y -619.236,Z 264.426,A 0.000,B 0.000,C 90.000,E1 292.642} C_DIS
LIN {X -0.042,Y -614.683,Z 264.416,A 0.000,B 0.000,C 90.000,E1 290.844} C_DIS
LIN {X -0.048,Y -610.387,Z 264.406,A 0.000,B 0.000,C 90.000,E1 289.033} C_DIS
LIN {X 0.084,Y -605.179,Z 264.393,A 0.000,B 0.000,C 90.000,E1 286.677} C_DIS
LIN {X -0.206,Y -602.055,Z 264.384,A 0.000,B 0.000,C 90.000,E1 285.134} C_DIS
LIN {X 0.062,Y -595.968,Z 264.364,A 0.000,B 0.000,C 90.000,E1 281.422} C_DIS
LIN {X 0.039,Y -594.606,Z 264.358,A 0.000,B 0.000,C 90.000,E1 280.366} C_DIS
LIN {X 0.296,Y -590.994,Z 264.339,A 0.000,B 0.000,C 90.000,E1 276.891} C_DIS
LIN {X -0.240,Y -589.135,Z 264.322,A 0.000,B 0.000,C 90.000,E1 274.012} C_DIS
LIN {X 0.198,Y -588.491,Z 264.310,A 0.000,B 0.000,C 90.000,E1 271.835} C_DIS
LIN {X 0.255,Y -588.740,Z 264.293,A 0.000,B 0.000,C 90.000,E1 268.625} C_DIS
LIN {X 0.236,Y -590.924,Z 264.272,A 0.000,B 0.000,C 90.000,E1 264.894} C_DIS
LIN {X 0.158,Y -593.637,Z 264.257,A 0.000,B 0.000,C 90.000,E1 262.243} C_DIS
LIN {X -0.262,Y -597.978,Z 264.239,A 0.000,B 0.000,C 90.000,E1 259.106} C_DIS
LIN {X -0.207,Y -601.284,Z 264.228,A 0.000,B 0.000,C 90.000,E1 256.992} C_DIS
LIN {X -0.146,Y -602.981,Z 264.222,A 0.000,B 0.000,C 90.000,E1 255.936} C_DIS
LIN {X -0.185,Y -604.929,Z 264.215,A 0.000,B 0.000,C 90.000,E1 254.629} C_DIS
LIN {X 0.074,Y -606.369,Z 264.209,A 0.000,B 0.000,C 90.000,E1 253.559} C_DIS
LIN {X 0.121,Y -606.958,Z 264.206,A 0.000,B 0.000,C 90.000,E1 253.032} C_DIS
LIN {X 0.265,Y -607.506,Z 264.202,A 0.000,B 0.000,C 90.000,E1 252.236} C_DIS
LIN {X -0.102,Y -608.164,Z 264.194,A 0.000,B 0.000,C 90.000,E1 250.967} C_DIS
LIN {X -0.132,Y -608.357,Z 264.190,A 0.000,B 0.000,C 90.000,E1 250.188} C_DIS
LIN {X 0.044,Y -608.381,Z 264.186,A 0.000,B 0.000,C 90.000,E1 249.390} C_DIS
LIN {X 0.221,Y -608.096,Z 264.181,A 0.000,B 0.000,C 90.000,E1 248.592} C_DIS
LIN {X -0.115,Y -607.823,Z 264.178,A 0.000,B 0.000,C 90.000,E1 248.103} C_DIS
LIN {X -0.003,Y -606.820,Z 264.173,A 0.000,B 0.000,C 90.000,E1 247.050} C_DIS
LIN {X 0.091,Y -605.552,Z 264.167,A 0.000,B 0.000,C 90.000,E1 245.997} C_DIS
LIN {X -0.138,Y -603.658,Z 264.161,A 0.000,B 0.000,C 90.000,E1 244.973} C_DIS
LIN {X 0.287,Y -602.587,Z 264.158,A 0.000,B 0.000,C 90.000,E1 244.409} C_DIS
LIN {X -0.044,Y -599.578,Z 264.151,A 0.000,B 0.000,C 90.000,E1 243.127} C_DIS
LIN {X -0.345,Y -596.965,Z 264.145,A 0.000,B 0.000,C 90.000,E1 242.103} C_DIS
LIN {X 0.315,Y -593.453,Z 264.138,A 0.000,B 0.000,C 90.000,E1 240.717} C_DIS
LIN {X 0.213,Y -590.549,Z 264.132,A 0.000,B 0.000,C 90.000,E1 239.665} C_DIS
LIN {X 0.064,Y -587.410,Z 264.126,A 0.000,B 0.000,C 90.000,E1 238.614} C_DIS
LIN {X 0.306,Y -584.919,Z 264.121,A 0.000,B 0.000,C 90.000,E1 237.788} C_DIS
LIN {X -0.085,Y -579.678,Z 264.112,A 0.000,B 0.000,C 90.000,E1 236.215} C_DIS
LIN {X 0.215,Y -574.521,Z 264.103,A 0.000,B 0.000,C 90.000,E1 234.562} C_DIS
LIN {X 0.129,Y -570.332,Z 264.096,A 0.000,B 0.000,C 90.000,E1 233.210} C_DIS
LIN {X -0.010,Y -565.316,Z 264.087,A 0.000,B 0.000,C 90.000,E1 231.582} C_DIS
LIN {X 0.192,Y -560.289,Z 264.077,A 0.000,B 0.000,C 90.000,E1 229.908} C_DIS
LIN {X 0.206,Y -555.119,Z 264.068,A 0.000,B 0.000,C 90.000,E1 228.243} C_DIS
LIN {X 0.052,Y -550.736,Z 264.060,A 0.000,B 0.000,C 90.000,E1 226.863} C_DIS
LIN {X -0.165,Y -544.519,Z 264.049,A 0.000,B 0.000,C 90.000,E1 224.919} C_DIS
LIN {X -0.145,Y -539.126,Z 264.040,A 0.000,B 0.000,C 90.000,E1 223.218} C_DIS
LIN {X 0.183,Y -534.692,Z 264.032,A 0.000,B 0.000,C 90.000,E1 221.757} C_DIS
LIN {X 0.083,Y -530.287,Z 264.024,A 0.000,B 0.000,C 90.000,E1 220.334} C_DIS
LIN {X 0.173,Y -524.190,Z 264.013,A 0.000,B 0.000,C 90.000,E1 218.302} C_DIS
LIN {X -0.193,Y -517.351,Z 264.000,A 0.000,B 0.000,C 90.000,E1 216.011} C_DIS
LIN {X 0.079,Y -510.664,Z 263.987,A 0.000,B 0.000,C 90.000,E1 213.627} C_DIS
LIN {X 0.010,Y -504.173,Z 263.974,A 0.000,B 0.000,C 90.000,E1 211.258} C_DIS
LIN {X 0.028,Y -499.595,Z 263.964,A 0.000,B 0.000,C 90.000,E1 209.461} C_DIS
LIN {X 0.035,Y -493.103,Z 263.949,A 0.000,B 0.000,C 90.000,E1 206.744} C_DIS
LIN {X -0.202,Y -488.489,Z 263.937,A 0.000,B 0.000,C 90.000,E1 204.643} C_DIS
LIN {X 0.139,Y -483.581,Z 263.923,A 0.000,B 0.000,C 90.000,E1 202.153} C_DIS
LIN {X 0.152,Y -479.594,Z 263.911,A 0.000,B 0.000,C 90.000,E1 199.993} C_DIS
LIN {X 0.182,Y -476.025,Z 263.899,A 0.000,B 0.000,C 90.000,E1 197.819} C_DIS
LIN {X 0.022,Y -473.177,Z 263.889,A 0.000,B 0.000,C 90.000,E1 195.969} C_DIS
LIN {X 0.074,Y -470.078,Z 263.877,A 0.000,B 0.000,C 90.000,E1 193.772} C_DIS
LIN {X 0.107,Y -467.759,Z 263.866,A 0.000,B 0.000,C 90.000,E1 191.883} C_DIS
LIN {X 0.151,Y -465.085,Z 263.854,A 0.000,B 0.000,C 90.000,E1 189.670} C_DIS
LIN {X -0.205,Y -463.043,Z 263.843,A 0.000,B 0.000,C 90.000,E1 187.814} C_DIS
LIN {X 0.222,Y -460.655,Z 263.829,A 0.000,B 0.000,C 90.000,E1 185.220} C_DIS
LIN {X 0.082,Y -459.079,Z 263.819,A 0.000,B 0.000,C 90.000,E1 183.326} C_DIS
LIN {X 0.019,Y -457.089,Z 263.803,A 0.000,B 0.000,C 90.000,E1 180.458} C_DIS
LIN {X -0.046,Y -455.791,Z 263.790,A 0.000,B 0.000,C 90.000,E1 178.224} C_DIS
LIN {X -0.123,Y -454.916,Z 263.778,A 0.000,B 0.000,C 90.000,E1 175.988} C_DIS
LIN {X -0.227,Y -454.337,Z 263.762,A 0.000,B 0.000,C 90.000,E1 173.109} C_DIS
LIN {X -0.145,Y -454.291,Z 263.749,A 0.000,B 0.000,C 90.000,E1 170.849} C_DIS
LIN {X 0.020,Y -454.543,Z 263.737,A 0.000,B 0.000,C 90.000,E1 168.578} C_DIS
LIN {X -0.150,Y -454.933,Z 263.728,A 0.000,B 0.000,C 90.000,E1 166.992} C_DIS
LIN {X 0.004,Y -455.506,Z 263.717,A 0.000,B 0.000,C 90.000,E1 165.046} C_DIS
LIN {X -0.062,Y -456.673,Z 263.703,A 0.000,B 0.000,C 90.000,E1 162.489} C_DIS
LIN {X -0.106,Y -458.436,Z 263.689,A 0.000,B 0.000,C 90.000,E1 159.934} C_DIS
LIN {X 0.073,Y -460.709,Z 263.674,A 0.000,B 0.000,C 90.000,E1 157.358} C_DIS
LIN {X -0.123,Y -464.141,Z 263.657,A 0.000,B 0.000,C 90.000,E1 154.204} C_DIS
LIN {X 0.069,Y -467.838,Z 263.641,A 0.000,B 0.000,C 90.000,E1 151.335} C_DIS
LIN {X -0.175,Y -472.098,Z 263.625,A 0.000,B 0.000,C 90.000,E1 148.535} C_DIS
LIN {X 0.054,Y -476.198,Z 263.611,A 0.000,B 0.000,C 90.000,E1 146.008} C_DIS
LIN {X -0.186,Y -478.818,Z 263.603,A 0.000,B 0.000,C 90.000,E1 144.482} C_DIS
LIN {X 0.000,Y -481.872,Z 263.592,A 0.000,B 0.000,C 90.000,E1 142.603} C_DIS
LIN {X -0.242,Y -484.218,Z 263.584,A 0.000,B 0.000,C 90.000,E1 141.090} C_DIS
LIN {X 0.032,Y -485.981,Z 263.577,A 0.000,B 0.000,C 90.000,E1 139.828} C_DIS
LIN {X -0.182,Y -487.196,Z 263.572,A 0.000,B 0.000,C 90.000,E1 138.933} C_DIS
LIN {X -0.062,Y -488.246,Z 263.567,A 0.000,B 0.000,C 90.000,E1 138.000} C_DIS
LIN {X 0.073,Y -489.143,Z 263.562,A 0.000,B 0.000,C 90.000,E1 137.067} C_DIS
LIN {X 0.056,Y -489.658,Z 263.558,A 0.000,B 0.000,C 90.000,E1 136.458} C_DIS
LIN {X -0.150,Y -490.168,Z 263.553,A 0.000,B 0.000,C 90.000,E1 135.567} C_DIS
LIN {X -0.182,Y -490.529,Z 263.546,A 0.000,B 0.000,C 90.000,E1 134.352} C_DIS
LIN {X 0.143,Y -490.588,Z 263.540,A 0.000,B 0.000,C 90.000,E1 133.095} C_DIS
LIN {X -0.058,Y -490.347,Z 263.534,A 0.000,B 0.000,C 90.000,E1 132.204} C_DIS
LIN {X -0.227,Y -489.870,Z 263.529,A 0.000,B 0.000,C 90.000,E1 131.310} C_DIS
LIN {X -0.079,Y -489.127,Z 263.524,A 0.000,B 0.000,C 90.000,E1 130.378} C_DIS
LIN {X 0.095,Y -487.508,Z 263.516,A 0.000,B 0.000,C 90.000,E1 128.830} C_DIS
LIN {X 0.111,Y -486.042,Z 263.509,A 0.000,B 0.000,C 90.000,E1 127.604} C_DIS
LIN {X 0.106,Y -484.344,Z 263.502,A 0.000,B 0.000,C 90.000,E1 126.377} C_DIS
LIN {X -0.032,Y -482.963,Z 263.497,A 0.000,B 0.000,C 90.000,E1 125.471} C_DIS
LIN {X -0.083,Y -479.761,Z 263.487,A 0.000,B 0.000,C 90.000,E1 123.627} C_DIS
LIN {X -0.079,Y -477.555,Z 263.480,A 0.000,B 0.000,C 90.000,E1 122.388} C_DIS
LIN {X 0.041,Y -475.359,Z 263.473,A 0.000,B 0.000,C 90.000,E1 121.131} C_DIS
LIN {X -0.151,Y -471.934,Z 263.463,A 0.000,B 0.000,C 90.000,E1 119.283} C_DIS
LIN {X -0.071,Y -467.962,Z 263.450,A 0.000,B 0.000,C 90.000,E1 117.078} C_DIS
LIN {X 0.240,Y -465.032,Z 263.442,A 0.000,B 0.000,C 90.000,E1 115.463} C_DIS
LIN {X 0.130,Y -461.030,Z 263.429,A 0.000,B 0.000,C 90.000,E1 113.259} C_DIS
LIN {X -0.018,Y -457.119,Z 263.417,A 0.000,B 0.000,C 90.000,E1 111.046} C_DIS
LIN {X 0.057,Y -455.874,Z 263.413,A 0.000,B 0.000,C 90.000,E1 110.301} C_DIS
LIN {X 0.017,Y -455.872,Z 263.413,A 0.000,B 0.000,C 90.000,E1 110.301} C_DIS
LIN {X 0.037,Y -457.354,Z 263.410,A 0.000,B 0.000,C 90.000,E1 109.758} C_DIS
LIN {X 0.122,Y -465.984,Z 263.387,A 0.000,B 0.000,C 90.000,E1 105.607} C_DIS
LIN {X -0.155,Y -467.550,Z 263.383,A 0.000,B 0.000,C 90.000,E1 105.009} C_DIS
LIN {X 0.028,Y -468.566,Z 263.380,A 0.000,B 0.000,C 90.000,E1 104.356} C_DIS
LIN {X -0.212,Y -475.786,Z 263.357,A 0.000,B 0.000,C 90.000,E1 100.310} C_DIS
LIN {X 0.093,Y -476.298,Z 263.355,A 0.000,B 0.000,C 90.000,E1 99.962} C_DIS
LIN {X 0.041,Y -481.777,Z 263.331,A 0.000,B 0.000,C 90.000,E1 95.625} C_DIS
LIN {X -0.112,Y -482.168,Z 263.330,A 0.000,B 0.000,C 90.000,E1 95.334} C_DIS
LIN {X -0.183,Y -485.300,Z 263.306,A 0.000,B 0.000,C 90.000,E1 91.031} C_DIS
LIN {X 0.127,Y -485.537,Z 263.304,A 0.000,B 0.000,C 90.000,E1 90.688} C_DIS
LIN {X -0.151,Y -486.316,Z 263.282,A 0.000,B 0.000,C 90.000,E1 86.731} C_DIS
LIN {X -0.016,Y -486.310,Z 263.278,A 0.000,B 0.000,C 90.000,E1 86.102} C_DIS
LIN {X 0.188,Y -484.696,Z 263.255,A 0.000,B 0.000,C 90.000,E1 81.781} C_DIS
LIN {X 0.057,Y -484.608,Z 263.253,A 0.000,B 0.000,C 90.000,E1 81.489} C_DIS
LIN {X -0.063,Y -480.540,Z 263.227,A 0.000,B 0.000,C 90.000,E1 76.881} C_DIS
LIN {X -0.152,Y -474.292,Z 263.201,A 0.000,B 0.000,C 90.000,E1 72.236} C_DIS
LIN {X 0.120,Y -473.863,Z 263.200,A 0.000,B 0.000,C 90.000,E1 71.891} C_DIS
LIN {X -0.146,Y -468.687,Z 263.184,A 0.000,B 0.000,C 90.000,E1 69.135} C_DIS
LIN {X 0.252,Y -468.683,Z 263.184,A 0.000,B 0.000,C 90.000,E1 69.082} C_DIS
LIN {X -0.251,Y -474.356,Z 263.172,A 0.000,B 0.000,C 90.000,E1 66.922} C_DIS
LIN {X -0.030,Y -480.091,Z 263.160,A 0.000,B 0.000,C 90.000,E1 64.717} C_DIS
LIN {X 0.125,Y -486.749,Z 263.146,A 0.000,B 0.000,C 90.000,E1 62.231} C_DIS
LIN {X -0.013,Y -490.983,Z 263.137,A 0.000,B 0.000,C 90.000,E1 60.717} C_DIS
LIN {X 0.048,Y -497.153,Z 263.126,A 0.000,B 0.000,C 90.000,E1 58.584} C_DIS
LIN {X -0.059,Y -501.485,Z 263.117,A 0.000,B 0.000,C 90.000,E1 57.089} C_DIS
LIN {X -0.092,Y -505.620,Z 263.109,A 0.000,B 0.000,C 90.000,E1 55.595} C_DIS
LIN {X -0.091,Y -508.762,Z 263.102,A 0.000,B 0.000,C 90.000,E1 54.402} C_DIS
LIN {X -0.132,Y -512.437,Z 263.094,A 0.000,B 0.000,C 90.000,E1 52.924} C_DIS
LIN {X -0.132,Y -515.147,Z 263.087,A 0.000,B 0.000,C 90.000,E1 51.743} C_DIS
LIN {X -0.087,Y -517.546,Z 263.081,A 0.000,B 0.000,C 90.000,E1 50.561} C_DIS
LIN {X 0.054,Y -519.234,Z 263.076,A 0.000,B 0.000,C 90.000,E1 49.666} C_DIS
LIN {X 0.151,Y -521.194,Z 263.070,A 0.000,B 0.000,C 90.000,E1 48.485} C_DIS
LIN {X 0.229,Y -522.788,Z 263.063,A 0.000,B 0.000,C 90.000,E1 47.310} C_DIS
LIN {X 0.030,Y -523.790,Z 263.058,A 0.000,B 0.000,C 90.000,E1 46.458} C_DIS
LIN {X 0.203,Y -524.585,Z 263.053,A 0.000,B 0.000,C 90.000,E1 45.567} C_DIS
LIN {X 0.015,Y -525.204,Z 263.048,A 0.000,B 0.000,C 90.000,E1 44.717} C_DIS
LIN {X 0.267,Y -525.558,Z 263.045,A 0.000,B 0.000,C 90.000,E1 44.109} C_DIS
LIN {X -0.021,Y -526.009,Z 263.037,A 0.000,B 0.000,C 90.000,E1 42.690} C_DIS
LIN {X 0.125,Y -526.139,Z 263.031,A 0.000,B 0.000,C 90.000,E1 41.515} C_DIS
LIN {X -0.043,Y -526.061,Z 263.026,A 0.000,B 0.000,C 90.000,E1 40.663} C_DIS
LIN {X -0.150,Y -525.803,Z 263.021,A 0.000,B 0.000,C 90.000,E1 39.806} C_DIS
LIN {X 0.014,Y -525.013,Z 263.013,A 0.000,B 0.000,C 90.000,E1 38.338} C_DIS
LIN {X 0.197,Y -524.174,Z 263.007,A 0.000,B 0.000,C 90.000,E1 37.156} C_DIS
LIN {X 0.084,Y -523.410,Z 263.002,A 0.000,B 0.000,C 90.000,E1 36.297} C_DIS
LIN {X -0.040,Y -522.462,Z 262.997,A 0.000,B 0.000,C 90.000,E1 35.438} C_DIS
LIN {X -0.195,Y -520.372,Z 262.987,A 0.000,B 0.000,C 90.000,E1 33.706} C_DIS
LIN {X -0.273,Y -518.832,Z 262.981,A 0.000,B 0.000,C 90.000,E1 32.546} C_DIS
LIN {X 0.015,Y -516.131,Z 262.969,A 0.000,B 0.000,C 90.000,E1 30.463} C_DIS
LIN {X 0.052,Y -514.664,Z 262.963,A 0.000,B 0.000,C 90.000,E1 29.283} C_DIS
LIN {X 0.067,Y -512.517,Z 262.953,A 0.000,B 0.000,C 90.000,E1 27.513} C_DIS
LIN {X -0.004,Y -509.744,Z 262.940,A 0.000,B 0.000,C 90.000,E1 25.155} C_DIS
LIN {X -0.103,Y -507.910,Z 262.930,A 0.000,B 0.000,C 90.000,E1 23.387} C_DIS
LIN {X 0.201,Y -505.513,Z 262.917,A 0.000,B 0.000,C 90.000,E1 20.972} C_DIS
LIN {X -0.008,Y -503.710,Z 262.905,A 0.000,B 0.000,C 90.000,E1 18.906} C_DIS
LIN {X 0.067,Y -502.458,Z 262.897,A 0.000,B 0.000,C 90.000,E1 17.402} C_DIS
LIN {X 0.052,Y -501.566,Z 262.890,A 0.000,B 0.000,C 90.000,E1 16.205} C_DIS
LIN {X -0.232,Y -499.685,Z 262.875,A 0.000,B 0.000,C 90.000,E1 13.536} C_DIS
LIN {X -0.243,Y -498.459,Z 262.862,A 0.000,B 0.000,C 90.000,E1 11.130} C_DIS
LIN {X 0.091,Y -497.657,Z 262.848,A 0.000,B 0.000,C 90.000,E1 8.681} C_DIS
LIN {X 0.174,Y -497.271,Z 262.835,A 0.000,B 0.000,C 90.000,E1 6.258} C_DIS
LIN {X 0.200,Y -497.289,Z 262.822,A 0.000,B 0.000,C 90.000,E1 3.841} C_DIS
LIN {X 0.158,Y -497.754,Z 262.808,A 0.000,B 0.000,C 90.000,E1 1.432} C_DIS
LIN {X -0.199,Y -498.906,Z 262.794,A 0.000,B 0.000,C 90.000,E1 358.912} C_DIS
LIN {X 0.194,Y -500.803,Z 262.779,A 0.000,B 0.000,C 90.000,E1 356.159} C_DIS
LIN {X -0.152,Y -502.984,Z 262.766,A 0.000,B 0.000,C 90.000,E1 353.799} C_DIS
LIN {X -0.037,Y -507.379,Z 262.747,A 0.000,B 0.000,C 90.000,E1 350.500} C_DIS
LIN {X 0.067,Y -511.443,Z 262.736,A 0.000,B 0.000,C 90.000,E1 348.409} C_DIS
LIN {X 0.054,Y -518.997,Z 262.719,A 0.000,B 0.000,C 90.000,E1 345.463} C_DIS
LIN {X -0.215,Y -523.647,Z 262.710,A 0.000,B 0.000,C 90.000,E1 343.740} C_DIS
LIN {X -0.055,Y -530.074,Z 262.697,A 0.000,B 0.000,C 90.000,E1 341.402} C_DIS
LIN {X -0.148,Y -538.120,Z 262.682,A 0.000,B 0.000,C 90.000,E1 338.827} C_DIS
LIN {X 0.009,Y -543.917,Z 262.673,A 0.000,B 0.000,C 90.000,E1 337.102} C_DIS
LIN {X -0.010,Y -547.811,Z 262.667,A 0.000,B 0.000,C 90.000,E1 335.973} C_DIS
LIN {X 0.111,Y -555.809,Z 262.654,A 0.000,B 0.000,C 90.000,E1 333.717} C_DIS
LIN {X 0.347,Y -562.018,Z 262.645,A 0.000,B 0.000,C 90.000,E1 332.025} C_DIS
LIN {X -0.246,Y -565.157,Z 262.640,A 0.000,B 0.000,C 90.000,E1 331.257} C_DIS
LIN {X 0.052,Y -569.215,Z 262.634,A 0.000,B 0.000,C 90.000,E1 330.127} C_DIS
LIN {X 0.243,Y -574.024,Z 262.627,A 0.000,B 0.000,C 90.000,E1 328.742} C_DIS
LIN {X -0.149,Y -582.724,Z 262.613,A 0.000,B 0.000,C 90.000,E1 326.342} C_DIS
LIN {X 0.285,Y -588.850,Z 262.604,A 0.000,B 0.000,C 90.000,E1 324.689} C_DIS
LIN {X 0.277,Y -592.855,Z 262.598,A 0.000,B 0.000,C 90.000,E1 323.623} C_DIS
LIN {X 0.079,Y -597.429,Z 262.591,A 0.000,B 0.000,C 90.000,E1 322.316} C_DIS
LIN {X 0.205,Y -602.679,Z 262.582,A 0.000,B 0.000,C 90.000,E1 320.723} C_DIS
LIN {X -0.304,Y -607.013,Z 262.575,A 0.000,B 0.000,C 90.000,E1 319.461} C_DIS
LIN {X 0.018,Y -613.958,Z 262.563,A 0.000,B 0.000,C 90.000,E1 317.349} C_DIS
LIN {X 0.216,Y -617.459,Z 262.557,A 0.000,B 0.000,C 90.000,E1 316.296} C_DIS
LIN {X 0.035,Y -620.634,Z 262.552,A 0.000,B 0.000,C 90.000,E1 315.283} C_DIS
LIN {X -0.107,Y -623.563,Z 262.546,A 0.000,B 0.000,C 90.000,E1 314.271} C_DIS
LIN {X 0.097,Y -626.988,Z 262.539,A 0.000,B 0.000,C 90.000,E1 312.975} C_DIS
LIN {X 0.043,Y -629.479,Z 262.533,A 0.000,B 0.000,C 90.000,E1 311.962} C_DIS
LIN {X -0.276,Y -631.127,Z 262.529,A 0.000,B 0.000,C 90.000,E1 311.229} C_DIS
LIN {X 0.205,Y -633.165,Z 262.523,A 0.000,B 0.000,C 90.000,E1 310.172} C_DIS
LIN {X -0.181,Y -634.915,Z 262.518,A 0.000,B 0.000,C 90.000,E1 309.197} C_DIS
LIN {X -0.053,Y -636.415,Z 262.512,A 0.000,B 0.000,C 90.000,E1 308.177} C_DIS
LIN {X 0.096,Y -637.708,Z 262.507,A 0.000,B 0.000,C 90.000,E1 307.156} C_DIS
LIN {X -0.122,Y -638.722,Z 262.501,A 0.000,B 0.000,C 90.000,E1 306.171} C_DIS
LIN {X 0.044,Y -639.227,Z 262.495,A 0.000,B 0.000,C 90.000,E1 305.152} C_DIS
LIN {X 0.367,Y -639.462,Z 262.490,A 0.000,B 0.000,C 90.000,E1 304.119} C_DIS
LIN {X 0.303,Y -639.526,Z 262.486,A 0.000,B 0.000,C 90.000,E1 303.372} C_DIS
LIN {X 0.244,Y -639.311,Z 262.481,A 0.000,B 0.000,C 90.000,E1 302.625} C_DIS
LIN {X 0.137,Y -639.056,Z 262.479,A 0.000,B 0.000,C 90.000,E1 302.133} C_DIS
LIN {X 0.115,Y -637.935,Z 262.473,A 0.000,B 0.000,C 90.000,E1 301.131} C_DIS
LIN {X -0.337,Y -637.194,Z 262.470,A 0.000,B 0.000,C 90.000,E1 300.669} C_DIS
LIN {X 0.171,Y -635.343,Z 262.465,A 0.000,B 0.000,C 90.000,E1 299.617} C_DIS
LIN {X 0.056,Y -633.710,Z 262.460,A 0.000,B 0.000,C 90.000,E1 298.871} C_DIS
LIN {X 0.243,Y -630.752,Z 262.453,A 0.000,B 0.000,C 90.000,E1 297.590} C_DIS
LIN {X -0.199,Y -628.142,Z 262.448,A 0.000,B 0.000,C 90.000,E1 296.616} C_DIS
LIN {X -0.103,Y -624.698,Z 262.441,A 0.000,B 0.000,C 90.000,E1 295.335} C_DIS
LIN {X 0.229,Y -619.960,Z 262.431,A 0.000,B 0.000,C 90.000,E1 293.515} C_DIS
LIN {X 0.203,Y -615.322,Z 262.421,A 0.000,B 0.000,C 90.000,E1 291.716} C_DIS
LIN {X 0.109,Y -609.708,Z 262.408,A 0.000,B 0.000,C 90.000,E1 289.396} C_DIS
LIN {X -0.089,Y -605.027,Z 262.396,A 0.000,B 0.000,C 90.000,E1 287.330} C_DIS
LIN {X 0.077,Y -601.266,Z 262.386,A 0.000,B 0.000,C 90.000,E1 285.481} C_DIS
LIN {X -0.015,Y -594.640,Z 262.364,A 0.000,B 0.000,C 90.000,E1 281.535} C_DIS
LIN {X 0.111,Y -592.898,Z 262.357,A 0.000,B 0.000,C 90.000,E1 280.197} C_DIS
LIN {X 0.125,Y -589.600,Z 262.339,A 0.000,B 0.000,C 90.000,E1 277.004} C_DIS
LIN {X -0.259,Y -587.329,Z 262.317,A 0.000,B 0.000,C 90.000,E1 273.037} C_DIS
LIN {X -0.073,Y -587.033,Z 262.297,A 0.000,B 0.000,C 90.000,E1 269.542} C_DIS
LIN {X -0.044,Y -588.418,Z 262.280,A 0.000,B 0.000,C 90.000,E1 266.331} C_DIS
LIN {X -0.272,Y -590.688,Z 262.265,A 0.000,B 0.000,C 90.000,E1 263.685} C_DIS
LIN {X 0.161,Y -592.778,Z 262.254,A 0.000,B 0.000,C 90.000,E1 261.781} C_DIS
LIN {X 0.110,Y -596.927,Z 262.238,A 0.000,B 0.000,C 90.000,E1 258.870} C_DIS
LIN {X 0.142,Y -600.253,Z 262.227,A 0.000,B 0.000,C 90.000,E1 256.756} C_DIS
LIN {X -0.090,Y -602.303,Z 262.219,A 0.000,B 0.000,C 90.000,E1 255.463} C_DIS
LIN {X -0.141,Y -604.180,Z 262.212,A 0.000,B 0.000,C 90.000,E1 254.157} C_DIS
LIN {X -0.205,Y -605.179,Z 262.208,A 0.000,B 0.000,C 90.000,E1 253.378} C_DIS
LIN {X 0.011,Y -605.704,Z 262.205,A 0.000,B 0.000,C 90.000,E1 252.834} C_DIS
LIN {X 0.272,Y -606.383,Z 262.199,A 0.000,B 0.000,C 90.000,E1 251.764} C_DIS
LIN {X -0.350,Y -606.745,Z 262.195,A 0.000,B 0.000,C 90.000,E1 251.040} C_DIS
LIN {X 0.309,Y -606.974,Z 262.189,A 0.000,B 0.000,C 90.000,E1 249.934} C_DIS
LIN {X -0.308,Y -606.885,Z 262.184,A 0.000,B 0.000,C 90.000,E1 249.209} C_DIS
LIN {X -0.208,Y -606.423,Z 262.179,A 0.000,B 0.000,C 90.000,E1 248.156} C_DIS
LIN {X -0.111,Y -605.433,Z 262.173,A 0.000,B 0.000,C 90.000,E1 247.102} C_DIS
LIN {X -0.032,Y -604.225,Z 262.167,A 0.000,B 0.000,C 90.000,E1 246.049} C_DIS
LIN {X 0.273,Y -602.303,Z 262.161,A 0.000,B 0.000,C 90.000,E1 244.973} C_DIS
LIN {X 0.145,Y -601.255,Z 262.158,A 0.000,B 0.000,C 90.000,E1 244.460} C_DIS
LIN {X 0.332,Y -598.249,Z 262.151,A 0.000,B 0.000,C 90.000,E1 243.127} C_DIS
LIN {X 0.011,Y -595.632,Z 262.145,A 0.000,B 0.000,C 90.000,E1 242.103} C_DIS
LIN {X -0.063,Y -592.838,Z 262.139,A 0.000,B 0.000,C 90.000,E1 241.051} C_DIS
LIN {X -0.283,Y -589.222,Z 262.132,A 0.000,B 0.000,C 90.000,E1 239.744} C_DIS
LIN {X -0.145,Y -586.046,Z 262.126,A 0.000,B 0.000,C 90.000,E1 238.663} C_DIS
LIN {X -0.223,Y -583.529,Z 262.121,A 0.000,B 0.000,C 90.000,E1 237.867} C_DIS
LIN {X -0.003,Y -579.159,Z 262.114,A 0.000,B 0.000,C 90.000,E1 236.501} C_DIS
LIN {X -0.188,Y -573.968,Z 262.105,A 0.000,B 0.000,C 90.000,E1 234.895} C_DIS
LIN {X -0.141,Y -568.914,Z 262.096,A 0.000,B 0.000,C 90.000,E1 233.256} C_DIS
LIN {X -0.205,Y -563.896,Z 262.087,A 0.000,B 0.000,C 90.000,E1 231.618} C_DIS
LIN {X 0.316,Y -558.850,Z 262.077,A 0.000,B 0.000,C 90.000,E1 229.908} C_DIS
LIN {X 0.298,Y -553.678,Z 262.068,A 0.000,B 0.000,C 90.000,E1 228.243} C_DIS
LIN {X 0.119,Y -549.281,Z 262.060,A 0.000,B 0.000,C 90.000,E1 226.863} C_DIS
LIN {X -0.136,Y -543.050,Z 262.050,A 0.000,B 0.000,C 90.000,E1 224.919} C_DIS
LIN {X -0.147,Y -537.632,Z 262.040,A 0.000,B 0.000,C 90.000,E1 223.218} C_DIS
LIN {X -0.194,Y -534.081,Z 262.034,A 0.000,B 0.000,C 90.000,E1 222.081} C_DIS
LIN {X 0.026,Y -528.796,Z 262.024,A 0.000,B 0.000,C 90.000,E1 220.334} C_DIS
LIN {X 0.079,Y -522.692,Z 262.013,A 0.000,B 0.000,C 90.000,E1 218.302} C_DIS
LIN {X 0.026,Y -515.056,Z 261.998,A 0.000,B 0.000,C 90.000,E1 215.678} C_DIS
LIN {X 0.233,Y -508.318,Z 261.985,A 0.000,B 0.000,C 90.000,E1 213.293} C_DIS
LIN {X 0.098,Y -501.901,Z 261.972,A 0.000,B 0.000,C 90.000,E1 210.924} C_DIS
LIN {X 0.212,Y -498.109,Z 261.964,A 0.000,B 0.000,C 90.000,E1 209.411} C_DIS
LIN {X -0.262,Y -491.620,Z 261.948,A 0.000,B 0.000,C 90.000,E1 206.744} C_DIS
LIN {X -0.090,Y -487.004,Z 261.937,A 0.000,B 0.000,C 90.000,E1 204.591} C_DIS
LIN {X -0.240,Y -482.718,Z 261.925,A 0.000,B 0.000,C 90.000,E1 202.461} C_DIS
LIN {X 0.192,Y -478.136,Z 261.911,A 0.000,B 0.000,C 90.000,E1 199.939} C_DIS
LIN {X -0.086,Y -475.120,Z 261.901,A 0.000,B 0.000,C 90.000,E1 198.109} C_DIS
LIN {X 0.179,Y -472.240,Z 261.890,A 0.000,B 0.000,C 90.000,E1 196.205} C_DIS
LIN {X -0.070,Y -469.568,Z 261.880,A 0.000,B 0.000,C 90.000,E1 194.356} C_DIS
LIN {X 0.216,Y -466.772,Z 261.868,A 0.000,B 0.000,C 90.000,E1 192.119} C_DIS
LIN {X -0.221,Y -464.104,Z 261.855,A 0.000,B 0.000,C 90.000,E1 189.962} C_DIS
LIN {X 0.113,Y -461.703,Z 261.843,A 0.000,B 0.000,C 90.000,E1 187.701} C_DIS
LIN {X -0.190,Y -459.618,Z 261.831,A 0.000,B 0.000,C 90.000,E1 185.511} C_DIS
LIN {X 0.142,Y -458.026,Z 261.820,A 0.000,B 0.000,C 90.000,E1 183.555} C_DIS
LIN {X 0.040,Y -455.981,Z 261.804,A 0.000,B 0.000,C 90.000,E1 180.688} C_DIS
LIN {X -0.055,Y -454.653,Z 261.791,A 0.000,B 0.000,C 90.000,E1 178.453} C_DIS
LIN {X 0.042,Y -453.631,Z 261.777,A 0.000,B 0.000,C 90.000,E1 175.869} C_DIS
LIN {X 0.061,Y -453.063,Z 261.759,A 0.000,B 0.000,C 90.000,E1 172.648} C_DIS
LIN {X 0.109,Y -453.101,Z 261.747,A 0.000,B 0.000,C 90.000,E1 170.387} C_DIS
LIN {X 0.024,Y -453.350,Z 261.736,A 0.000,B 0.000,C 90.000,E1 168.465} C_DIS
LIN {X -0.173,Y -453.780,Z 261.727,A 0.000,B 0.000,C 90.000,E1 166.881} C_DIS
LIN {X -0.053,Y -454.383,Z 261.716,A 0.000,B 0.000,C 90.000,E1 164.936} C_DIS
LIN {X -0.028,Y -455.584,Z 261.702,A 0.000,B 0.000,C 90.000,E1 162.362} C_DIS
LIN {X -0.004,Y -457.161,Z 261.690,A 0.000,B 0.000,C 90.000,E1 160.115} C_DIS
LIN {X 0.139,Y -459.376,Z 261.675,A 0.000,B 0.000,C 90.000,E1 157.539} C_DIS
LIN {X 0.277,Y -461.976,Z 261.661,A 0.000,B 0.000,C 90.000,E1 154.973} C_DIS
LIN {X 0.160,Y -463.538,Z 261.654,A 0.000,B 0.000,C 90.000,E1 153.717} C_DIS
LIN {X 0.203,Y -466.914,Z 261.640,A 0.000,B 0.000,C 90.000,E1 151.179} C_DIS
LIN {X 0.181,Y -470.709,Z 261.626,A 0.000,B 0.000,C 90.000,E1 148.663} C_DIS
LIN {X 0.110,Y -474.769,Z 261.612,A 0.000,B 0.000,C 90.000,E1 146.167} C_DIS
LIN {X 0.319,Y -476.890,Z 261.605,A 0.000,B 0.000,C 90.000,E1 144.895} C_DIS
LIN {X -0.101,Y -478.911,Z 261.598,A 0.000,B 0.000,C 90.000,E1 143.703} C_DIS
LIN {X -0.210,Y -480.940,Z 261.591,A 0.000,B 0.000,C 90.000,E1 142.477} C_DIS
LIN {X 0.204,Y -483.258,Z 261.583,A 0.000,B 0.000,C 90.000,E1 140.884} C_DIS
LIN {X -0.090,Y -485.407,Z 261.574,A 0.000,B 0.000,C 90.000,E1 139.380} C_DIS
LIN {X -0.169,Y -486.871,Z 261.568,A 0.000,B 0.000,C 90.000,E1 138.162} C_DIS
LIN {X -0.052,Y -487.789,Z 261.562,A 0.000,B 0.000,C 90.000,E1 137.229} C_DIS
LIN {X 0.076,Y -488.495,Z 261.557,A 0.000,B 0.000,C 90.000,E1 136.296} C_DIS
LIN {X -0.142,Y -488.987,Z 261.552,A 0.000,B 0.000,C 90.000,E1 135.405} C_DIS
LIN {X -0.192,Y -489.328,Z 261.545,A 0.000,B 0.000,C 90.000,E1 134.190} C_DIS
LIN {X -0.047,Y -489.404,Z 261.540,A 0.000,B 0.000,C 90.000,E1 133.257} C_DIS
LIN {X 0.102,Y -489.202,Z 261.535,A 0.000,B 0.000,C 90.000,E1 132.324} C_DIS
LIN {X -0.118,Y -488.762,Z 261.530,A 0.000,B 0.000,C 90.000,E1 131.434} C_DIS
LIN {X 0.217,Y -487.765,Z 261.523,A 0.000,B 0.000,C 90.000,E1 130.172} C_DIS
LIN {X -0.009,Y -486.176,Z 261.515,A 0.000,B 0.000,C 90.000,E1 128.669} C_DIS
LIN {X -0.016,Y -484.703,Z 261.508,A 0.000,B 0.000,C 90.000,E1 127.443} C_DIS
LIN {X -0.046,Y -482.998,Z 261.501,A 0.000,B 0.000,C 90.000,E1 126.217} C_DIS
LIN {X -0.202,Y -481.569,Z 261.496,A 0.000,B 0.000,C 90.000,E1 125.311} C_DIS
LIN {X 0.109,Y -478.410,Z 261.486,A 0.000,B 0.000,C 90.000,E1 123.420} C_DIS
LIN {X -0.185,Y -475.139,Z 261.475,A 0.000,B 0.000,C 90.000,E1 121.592} C_DIS
LIN {X 0.083,Y -472.295,Z 261.467,A 0.000,B 0.000,C 90.000,E1 120.001} C_DIS
LIN {X 0.068,Y -469.433,Z 261.458,A 0.000,B 0.000,C 90.000,E1 118.437} C_DIS
LIN {X -0.065,Y -466.047,Z 261.448,A 0.000,B 0.000,C 90.000,E1 116.565} C_DIS
LIN {X 0.009,Y -463.117,Z 261.439,A 0.000,B 0.000,C 90.000,E1 114.975} C_DIS
LIN {X -0.061,Y -459.715,Z 261.428,A 0.000,B 0.000,C 90.000,E1 113.078} C_DIS
LIN {X -0.075,Y -455.846,Z 261.416,A 0.000,B 0.000,C 90.000,E1 110.844} C_DIS
LIN {X 0.255,Y -455.301,Z 261.414,A 0.000,B 0.000,C 90.000,E1 110.482} C_DIS
LIN {X 0.215,Y -455.302,Z 261.414,A 0.000,B 0.000,C 90.000,E1 110.482} C_DIS
LIN {X -0.098,Y -457.085,Z 261.410,A 0.000,B 0.000,C 90.000,E1 109.885} C_DIS
LIN {X 0.120,Y -462.804,Z 261.395,A 0.000,B 0.000,C 90.000,E1 106.985} C_DIS
LIN {X 0.158,Y -467.276,Z 261.384,A 0.000,B 0.000,C 90.000,E1 105.079} C_DIS
LIN {X 0.083,Y -467.966,Z 261.382,A 0.000,B 0.000,C 90.000,E1 104.773} C_DIS
LIN {X 0.047,Y -476.184,Z 261.356,A 0.000,B 0.000,C 90.000,E1 100.074} C_DIS
LIN {X -0.178,Y -482.090,Z 261.330,A 0.000,B 0.000,C 90.000,E1 95.448} C_DIS
LIN {X 0.052,Y -485.506,Z 261.305,A 0.000,B 0.000,C 90.000,E1 90.802} C_DIS
LIN {X 0.085,Y -486.384,Z 261.281,A 0.000,B 0.000,C 90.000,E1 86.502} C_DIS
LIN {X -0.091,Y -486.361,Z 261.279,A 0.000,B 0.000,C 90.000,E1 86.216} C_DIS
LIN {X -0.007,Y -484.684,Z 261.253,A 0.000,B 0.000,C 90.000,E1 81.602} C_DIS
LIN {X -0.108,Y -480.605,Z 261.228,A 0.000,B 0.000,C 90.000,E1 76.992} C_DIS
LIN {X 0.217,Y -480.240,Z 261.226,A 0.000,B 0.000,C 90.000,E1 76.645} C_DIS
LIN {X 0.106,Y -474.070,Z 261.200,A 0.000,B 0.000,C 90.000,E1 72.000} C_DIS
LIN {X -0.114,Y -468.314,Z 261.183,A 0.000,B 0.000,C 90.000,E1 68.901} C_DIS
LIN {X -0.154,Y -468.311,Z 261.183,A 0.000,B 0.000,C 90.000,E1 68.901} C_DIS
LIN {X 0.022,Y -474.261,Z 261.170,A 0.000,B 0.000,C 90.000,E1 66.561} C_DIS
LIN {X -0.182,Y -479.171,Z 261.159,A 0.000,B 0.000,C 90.000,E1 64.717} C_DIS
LIN {X -0.053,Y -484.951,Z 261.147,A 0.000,B 0.000,C 90.000,E1 62.538} C_DIS
LIN {X 0.211,Y -490.021,Z 261.137,A 0.000,B 0.000,C 90.000,E1 60.667} C_DIS
LIN {X -0.029,Y -495.279,Z 261.127,A 0.000,B 0.000,C 90.000,E1 58.869} C_DIS
LIN {X 0.110,Y -500.494,Z 261.117,A 0.000,B 0.000,C 90.000,E1 57.041} C_DIS
LIN {X 0.052,Y -504.588,Z 261.109,A 0.000,B 0.000,C 90.000,E1 55.548} C_DIS
LIN {X 0.033,Y -507.718,Z 261.102,A 0.000,B 0.000,C 90.000,E1 54.356} C_DIS
LIN {X -0.046,Y -510.677,Z 261.095,A 0.000,B 0.000,C 90.000,E1 53.176} C_DIS
LIN {X -0.056,Y -514.057,Z 261.087,A 0.000,B 0.000,C 90.000,E1 51.698} C_DIS
LIN {X -0.105,Y -517.047,Z 261.079,A 0.000,B 0.000,C 90.000,E1 50.231} C_DIS
LIN {X -0.097,Y -519.116,Z 261.073,A 0.000,B 0.000,C 90.000,E1 49.057} C_DIS
LIN {X -0.007,Y -520.867,Z 261.066,A 0.000,B 0.000,C 90.000,E1 47.877} C_DIS
LIN {X 0.065,Y -522.312,Z 261.060,A 0.000,B 0.000,C 90.000,E1 46.701} C_DIS
LIN {X 0.219,Y -523.155,Z 261.055,A 0.000,B 0.000,C 90.000,E1 45.810} C_DIS
LIN {X -0.049,Y -523.980,Z 261.048,A 0.000,B 0.000,C 90.000,E1 44.676} C_DIS
LIN {X 0.126,Y -524.398,Z 261.043,A 0.000,B 0.000,C 90.000,E1 43.785} C_DIS
LIN {X 0.252,Y -524.746,Z 261.037,A 0.000,B 0.000,C 90.000,E1 42.609} C_DIS
LIN {X 0.030,Y -524.845,Z 261.030,A 0.000,B 0.000,C 90.000,E1 41.472} C_DIS
LIN {X -0.146,Y -524.743,Z 261.026,A 0.000,B 0.000,C 90.000,E1 40.620} C_DIS
LIN {X 0.073,Y -524.451,Z 261.021,A 0.000,B 0.000,C 90.000,E1 39.725} C_DIS
LIN {X 0.250,Y -523.825,Z 261.014,A 0.000,B 0.000,C 90.000,E1 38.543} C_DIS
LIN {X 0.095,Y -523.029,Z 261.008,A 0.000,B 0.000,C 90.000,E1 37.397} C_DIS
LIN {X 0.241,Y -521.980,Z 261.001,A 0.000,B 0.000,C 90.000,E1 36.217} C_DIS
LIN {X -0.250,Y -520.640,Z 260.995,A 0.000,B 0.000,C 90.000,E1 35.105} C_DIS
LIN {X -0.092,Y -518.844,Z 260.987,A 0.000,B 0.000,C 90.000,E1 33.627} C_DIS
LIN {X 0.240,Y -517.243,Z 260.980,A 0.000,B 0.000,C 90.000,E1 32.418} C_DIS
LIN {X 0.140,Y -514.154,Z 260.967,A 0.000,B 0.000,C 90.000,E1 30.079} C_DIS
LIN {X 0.041,Y -511.569,Z 260.956,A 0.000,B 0.000,C 90.000,E1 28.025} C_DIS
LIN {X 0.198,Y -509.403,Z 260.946,A 0.000,B 0.000,C 90.000,E1 26.232} C_DIS
LIN {X -0.177,Y -506.833,Z 260.933,A 0.000,B 0.000,C 90.000,E1 23.898} C_DIS
LIN {X 0.027,Y -505.288,Z 260.924,A 0.000,B 0.000,C 90.000,E1 22.386} C_DIS
LIN {X -0.017,Y -503.303,Z 260.913,A 0.000,B 0.000,C 90.000,E1 20.301} C_DIS
LIN {X 0.195,Y -501.548,Z 260.901,A 0.000,B 0.000,C 90.000,E1 18.181} C_DIS
LIN {X 0.204,Y -499.882,Z 260.889,A 0.000,B 0.000,C 90.000,E1 16.079} C_DIS
LIN {X -0.065,Y -498.195,Z 260.876,A 0.000,B 0.000,C 90.000,E1 13.703} C_DIS
LIN {X -0.051,Y -497.069,Z 260.864,A 0.000,B 0.000,C 90.000,E1 11.591} C_DIS
LIN {X 0.064,Y -496.062,Z 260.849,A 0.000,B 0.000,C 90.000,E1 8.859} C_DIS
LIN {X -0.228,Y -495.667,Z 260.838,A 0.000,B 0.000,C 90.000,E1 6.777} C_DIS
LIN {X 0.138,Y -495.600,Z 260.822,A 0.000,B 0.000,C 90.000,E1 4.012} C_DIS
LIN {X 0.165,Y -495.913,Z 260.811,A 0.000,B 0.000,C 90.000,E1 1.892} C_DIS
LIN {X -0.217,Y -497.183,Z 260.794,A 0.000,B 0.000,C 90.000,E1 358.912} C_DIS
LIN {X 0.017,Y -499.301,Z 260.777,A 0.000,B 0.000,C 90.000,E1 355.869} C_DIS
LIN {X 0.216,Y -502.966,Z 260.757,A 0.000,B 0.000,C 90.000,E1 352.243} C_DIS
LIN {X 0.007,Y -507.220,Z 260.742,A 0.000,B 0.000,C 90.000,E1 349.577} C_DIS
LIN {X -0.160,Y -511.122,Z 260.732,A 0.000,B 0.000,C 90.000,E1 347.813} C_DIS
LIN {X -0.283,Y -518.092,Z 260.717,A 0.000,B 0.000,C 90.000,E1 345.172} C_DIS
LIN {X 0.068,Y -522.796,Z 260.708,A 0.000,B 0.000,C 90.000,E1 343.378} C_DIS
LIN {X 0.208,Y -529.301,Z 260.695,A 0.000,B 0.000,C 90.000,E1 341.040} C_DIS
LIN {X -0.117,Y -536.551,Z 260.682,A 0.000,B 0.000,C 90.000,E1 338.773} C_DIS
LIN {X 0.000,Y -542.361,Z 260.673,A 0.000,B 0.000,C 90.000,E1 337.050} C_DIS
LIN {X -0.046,Y -546.268,Z 260.666,A 0.000,B 0.000,C 90.000,E1 335.921} C_DIS
LIN {X 0.266,Y -554.282,Z 260.654,A 0.000,B 0.000,C 90.000,E1 333.640} C_DIS
LIN {X 0.214,Y -560.499,Z 260.644,A 0.000,B 0.000,C 90.000,E1 331.975} C_DIS
LIN {X -0.127,Y -563.652,Z 260.640,A 0.000,B 0.000,C 90.000,E1 331.179} C_DIS
LIN {X -0.129,Y -567.722,Z 260.634,A 0.000,B 0.000,C 90.000,E1 330.078} C_DIS
LIN {X 0.325,Y -572.550,Z 260.626,A 0.000,B 0.000,C 90.000,E1 328.663} C_DIS
LIN {X 0.380,Y -581.328,Z 260.613,A 0.000,B 0.000,C 90.000,E1 326.215} C_DIS
LIN {X 0.115,Y -586.491,Z 260.605,A 0.000,B 0.000,C 90.000,E1 324.895} C_DIS
LIN {X -0.071,Y -591.447,Z 260.598,A 0.000,B 0.000,C 90.000,E1 323.577} C_DIS
LIN {X -0.304,Y -595.998,Z 260.590,A 0.000,B 0.000,C 90.000,E1 322.271} C_DIS
LIN {X 0.159,Y -601.267,Z 260.581,A 0.000,B 0.000,C 90.000,E1 320.642} C_DIS
LIN {X 0.087,Y -605.655,Z 260.574,A 0.000,B 0.000,C 90.000,E1 319.337} C_DIS
LIN {X -0.356,Y -611.788,Z 260.564,A 0.000,B 0.000,C 90.000,E1 317.553} C_DIS
LIN {X 0.261,Y -615.404,Z 260.558,A 0.000,B 0.000,C 90.000,E1 316.458} C_DIS
LIN {X -0.230,Y -617.885,Z 260.554,A 0.000,B 0.000,C 90.000,E1 315.729} C_DIS
LIN {X 0.032,Y -620.970,Z 260.548,A 0.000,B 0.000,C 90.000,E1 314.676} C_DIS
LIN {X 0.195,Y -624.436,Z 260.541,A 0.000,B 0.000,C 90.000,E1 313.380} C_DIS
LIN {X 0.112,Y -627.021,Z 260.535,A 0.000,B 0.000,C 90.000,E1 312.366} C_DIS
LIN {X 0.060,Y -629.339,Z 260.530,A 0.000,B 0.000,C 90.000,E1 311.353} C_DIS
LIN {X -0.022,Y -631.825,Z 260.523,A 0.000,B 0.000,C 90.000,E1 310.092} C_DIS
LIN {X 0.096,Y -633.143,Z 260.519,A 0.000,B 0.000,C 90.000,E1 309.322} C_DIS
LIN {X 0.195,Y -634.662,Z 260.513,A 0.000,B 0.000,C 90.000,E1 308.302} C_DIS
LIN {X -0.070,Y -635.951,Z 260.507,A 0.000,B 0.000,C 90.000,E1 307.317} C_DIS
LIN {X 0.071,Y -636.980,Z 260.502,A 0.000,B 0.000,C 90.000,E1 306.297} C_DIS
LIN {X 0.344,Y -637.459,Z 260.498,A 0.000,B 0.000,C 90.000,E1 305.518} C_DIS
LIN {X -0.268,Y -637.701,Z 260.493,A 0.000,B 0.000,C 90.000,E1 304.818} C_DIS
LIN {X 0.424,Y -637.888,Z 260.486,A 0.000,B 0.000,C 90.000,E1 303.499} C_DIS
LIN {X 0.345,Y -637.712,Z 260.482,A 0.000,B 0.000,C 90.000,E1 302.752} C_DIS
LIN {X 0.267,Y -637.255,Z 260.478,A 0.000,B 0.000,C 90.000,E1 302.005} C_DIS
LIN {X 0.224,Y -636.115,Z 260.472,A 0.000,B 0.000,C 90.000,E1 301.003} C_DIS
LIN {X 0.125,Y -634.887,Z 260.468,A 0.000,B 0.000,C 90.000,E1 300.256} C_DIS
LIN {X -0.306,Y -633.427,Z 260.464,A 0.000,B 0.000,C 90.000,E1 299.539} C_DIS
LIN {X 0.145,Y -631.212,Z 260.458,A 0.000,B 0.000,C 90.000,E1 298.487} C_DIS
LIN {X -0.266,Y -628.173,Z 260.451,A 0.000,B 0.000,C 90.000,E1 297.257} C_DIS
LIN {X -0.167,Y -624.789,Z 260.444,A 0.000,B 0.000,C 90.000,E1 295.976} C_DIS
LIN {X 0.172,Y -619.950,Z 260.434,A 0.000,B 0.000,C 90.000,E1 294.155} C_DIS
LIN {X -0.152,Y -615.967,Z 260.426,A 0.000,B 0.000,C 90.000,E1 292.642} C_DIS
LIN {X 0.298,Y -611.432,Z 260.416,A 0.000,B 0.000,C 90.000,E1 290.791} C_DIS
LIN {X -0.156,Y -607.167,Z 260.406,A 0.000,B 0.000,C 90.000,E1 289.014} C_DIS
LIN {X -0.043,Y -602.530,Z 260.394,A 0.000,B 0.000,C 90.000,E1 286.913} C_DIS
LIN {X 0.190,Y -599.391,Z 260.385,A 0.000,B 0.000,C 90.000,E1 285.315} C_DIS
LIN {X 0.176,Y -593.597,Z 260.366,A 0.000,B 0.000,C 90.000,E1 281.883} C_DIS
LIN {X -0.031,Y -591.502,Z 260.357,A 0.000,B 0.000,C 90.000,E1 280.310} C_DIS
LIN {X 0.092,Y -587.914,Z 260.338,A 0.000,B 0.000,C 90.000,E1 276.834} C_DIS
LIN {X 0.215,Y -585.957,Z 260.320,A 0.000,B 0.000,C 90.000,E1 273.612} C_DIS
LIN {X -0.183,Y -585.457,Z 260.310,A 0.000,B 0.000,C 90.000,E1 271.776} C_DIS
LIN {X -0.082,Y -585.877,Z 260.290,A 0.000,B 0.000,C 90.000,E1 268.282} C_DIS
LIN {X -0.033,Y -587.903,Z 260.273,A 0.000,B 0.000,C 90.000,E1 265.065} C_DIS
LIN {X -0.027,Y -590.947,Z 260.256,A 0.000,B 0.000,C 90.000,E1 262.129} C_DIS
LIN {X 0.131,Y -595.385,Z 260.239,A 0.000,B 0.000,C 90.000,E1 258.926} C_DIS
LIN {X -0.012,Y -598.684,Z 260.227,A 0.000,B 0.000,C 90.000,E1 256.825} C_DIS
LIN {X -0.129,Y -600.724,Z 260.220,A 0.000,B 0.000,C 90.000,E1 255.519} C_DIS
LIN {X 0.073,Y -602.276,Z 260.214,A 0.000,B 0.000,C 90.000,E1 254.448} C_DIS
LIN {X 0.296,Y -603.633,Z 260.208,A 0.000,B 0.000,C 90.000,E1 253.378} C_DIS
LIN {X 0.228,Y -604.376,Z 260.203,A 0.000,B 0.000,C 90.000,E1 252.598} C_DIS
LIN {X -0.108,Y -605.014,Z 260.198,A 0.000,B 0.000,C 90.000,E1 251.583} C_DIS
LIN {X -0.248,Y -605.390,Z 260.192,A 0.000,B 0.000,C 90.000,E1 250.550} C_DIS
LIN {X 0.183,Y -605.456,Z 260.186,A 0.000,B 0.000,C 90.000,E1 249.464} C_DIS
LIN {X -0.240,Y -605.230,Z 260.182,A 0.000,B 0.000,C 90.000,E1 248.720} C_DIS
LIN {X -0.098,Y -604.745,Z 260.177,A 0.000,B 0.000,C 90.000,E1 247.922} C_DIS
LIN {X -0.032,Y -603.694,Z 260.172,A 0.000,B 0.000,C 90.000,E1 246.869} C_DIS
LIN {X -0.225,Y -602.743,Z 260.167,A 0.000,B 0.000,C 90.000,E1 246.102} C_DIS
LIN {X -0.189,Y -600.882,Z 260.161,A 0.000,B 0.000,C 90.000,E1 245.049} C_DIS
LIN {X -0.329,Y -599.841,Z 260.158,A 0.000,B 0.000,C 90.000,E1 244.537} C_DIS
LIN {X 0.099,Y -596.842,Z 260.151,A 0.000,B 0.000,C 90.000,E1 243.179} C_DIS
LIN {X -0.233,Y -594.237,Z 260.145,A 0.000,B 0.000,C 90.000,E1 242.153} C_DIS
LIN {X 0.196,Y -591.462,Z 260.139,A 0.000,B 0.000,C 90.000,E1 241.051} C_DIS
LIN {X -0.046,Y -587.821,Z 260.132,A 0.000,B 0.000,C 90.000,E1 239.744} C_DIS
LIN {X 0.069,Y -584.638,Z 260.126,A 0.000,B 0.000,C 90.000,E1 238.663} C_DIS
LIN {X -0.024,Y -582.089,Z 260.122,A 0.000,B 0.000,C 90.000,E1 237.867} C_DIS
LIN {X 0.169,Y -577.700,Z 260.114,A 0.000,B 0.000,C 90.000,E1 236.501} C_DIS
LIN {X 0.095,Y -571.642,Z 260.103,A 0.000,B 0.000,C 90.000,E1 234.609} C_DIS
LIN {X -0.032,Y -567.447,Z 260.096,A 0.000,B 0.000,C 90.000,E1 233.256} C_DIS
LIN {X -0.127,Y -562.393,Z 260.087,A 0.000,B 0.000,C 90.000,E1 231.618} C_DIS
LIN {X 0.359,Y -557.332,Z 260.078,A 0.000,B 0.000,C 90.000,E1 229.908} C_DIS
LIN {X 0.309,Y -552.161,Z 260.068,A 0.000,B 0.000,C 90.000,E1 228.243} C_DIS
LIN {X 0.103,Y -547.746,Z 260.060,A 0.000,B 0.000,C 90.000,E1 226.863} C_DIS
LIN {X 0.190,Y -542.383,Z 260.051,A 0.000,B 0.000,C 90.000,E1 225.162} C_DIS
LIN {X -0.203,Y -537.863,Z 260.043,A 0.000,B 0.000,C 90.000,E1 223.785} C_DIS
LIN {X 0.104,Y -533.418,Z 260.035,A 0.000,B 0.000,C 90.000,E1 222.324} C_DIS
LIN {X -0.090,Y -528.087,Z 260.026,A 0.000,B 0.000,C 90.000,E1 220.620} C_DIS
LIN {X -0.057,Y -521.973,Z 260.014,A 0.000,B 0.000,C 90.000,E1 218.588} C_DIS
LIN {X -0.006,Y -515.960,Z 260.003,A 0.000,B 0.000,C 90.000,E1 216.537} C_DIS
LIN {X 0.021,Y -512.621,Z 259.996,A 0.000,B 0.000,C 90.000,E1 215.358} C_DIS
LIN {X -0.039,Y -506.747,Z 259.985,A 0.000,B 0.000,C 90.000,E1 213.293} C_DIS
LIN {X -0.216,Y -500.332,Z 259.972,A 0.000,B 0.000,C 90.000,E1 210.924} C_DIS
LIN {X -0.130,Y -496.518,Z 259.963,A 0.000,B 0.000,C 90.000,E1 209.411} C_DIS
LIN {X -0.239,Y -490.725,Z 259.950,A 0.000,B 0.000,C 90.000,E1 207.001} C_DIS
LIN {X 0.139,Y -484.823,Z 259.935,A 0.000,B 0.000,C 90.000,E1 204.207} C_DIS
LIN {X -0.075,Y -481.148,Z 259.924,A 0.000,B 0.000,C 90.000,E1 202.386} C_DIS
LIN {X 0.150,Y -477.197,Z 259.912,A 0.000,B 0.000,C 90.000,E1 200.194} C_DIS
LIN {X 0.242,Y -473.124,Z 259.898,A 0.000,B 0.000,C 90.000,E1 197.692} C_DIS
LIN {X 0.011,Y -470.284,Z 259.888,A 0.000,B 0.000,C 90.000,E1 195.843} C_DIS
LIN {X 0.055,Y -467.686,Z 259.878,A 0.000,B 0.000,C 90.000,E1 193.953} C_DIS
LIN {X -0.156,Y -464.974,Z 259.865,A 0.000,B 0.000,C 90.000,E1 191.771} C_DIS
LIN {X -0.179,Y -462.317,Z 259.853,A 0.000,B 0.000,C 90.000,E1 189.557} C_DIS
LIN {X 0.107,Y -459.995,Z 259.841,A 0.000,B 0.000,C 90.000,E1 187.296} C_DIS
LIN {X 0.213,Y -457.964,Z 259.828,A 0.000,B 0.000,C 90.000,E1 185.049} C_DIS
LIN {X -0.050,Y -455.894,Z 259.814,A 0.000,B 0.000,C 90.000,E1 182.522} C_DIS
LIN {X 0.139,Y -454.606,Z 259.803,A 0.000,B 0.000,C 90.000,E1 180.573} C_DIS
LIN {X 0.007,Y -453.287,Z 259.791,A 0.000,B 0.000,C 90.000,E1 178.339} C_DIS
LIN {X 0.059,Y -452.293,Z 259.777,A 0.000,B 0.000,C 90.000,E1 175.755} C_DIS
LIN {X -0.122,Y -451.786,Z 259.760,A 0.000,B 0.000,C 90.000,E1 172.875} C_DIS
LIN {X -0.173,Y -451.827,Z 259.748,A 0.000,B 0.000,C 90.000,E1 170.622} C_DIS
LIN {X 0.241,Y -452.068,Z 259.737,A 0.000,B 0.000,C 90.000,E1 168.634} C_DIS
LIN {X -0.074,Y -452.512,Z 259.728,A 0.000,B 0.000,C 90.000,E1 167.061} C_DIS
LIN {X 0.129,Y -453.135,Z 259.717,A 0.000,B 0.000,C 90.000,E1 165.102} C_DIS
LIN {X -0.003,Y -454.304,Z 259.703,A 0.000,B 0.000,C 90.000,E1 162.543} C_DIS
LIN {X -0.015,Y -455.883,Z 259.691,A 0.000,B 0.000,C 90.000,E1 160.296} C_DIS
LIN {X 0.090,Y -458.028,Z 259.676,A 0.000,B 0.000,C 90.000,E1 157.720} C_DIS
LIN {X 0.084,Y -460.314,Z 259.664,A 0.000,B 0.000,C 90.000,E1 155.485} C_DIS
LIN {X -0.025,Y -462.576,Z 259.653,A 0.000,B 0.000,C 90.000,E1 153.589} C_DIS
LIN {X -0.012,Y -465.998,Z 259.639,A 0.000,B 0.000,C 90.000,E1 151.051} C_DIS
LIN {X -0.066,Y -469.790,Z 259.625,A 0.000,B 0.000,C 90.000,E1 148.535} C_DIS
LIN {X 0.092,Y -473.900,Z 259.611,A 0.000,B 0.000,C 90.000,E1 146.008} C_DIS
LIN {X -0.190,Y -476.516,Z 259.603,A 0.000,B 0.000,C 90.000,E1 144.482} C_DIS
LIN {X -0.060,Y -479.506,Z 259.592,A 0.000,B 0.000,C 90.000,E1 142.603} C_DIS
LIN {X 0.030,Y -481.835,Z 259.584,A 0.000,B 0.000,C 90.000,E1 141.045} C_DIS
LIN {X 0.020,Y -483.972,Z 259.575,A 0.000,B 0.000,C 90.000,E1 139.504} C_DIS
LIN {X 0.150,Y -485.084,Z 259.570,A 0.000,B 0.000,C 90.000,E1 138.566} C_DIS
LIN {X -0.115,Y -486.106,Z 259.565,A 0.000,B 0.000,C 90.000,E1 137.676} C_DIS
LIN {X -0.188,Y -487.137,Z 259.558,A 0.000,B 0.000,C 90.000,E1 136.458} C_DIS
LIN {X -0.267,Y -487.775,Z 259.551,A 0.000,B 0.000,C 90.000,E1 135.243} C_DIS
LIN {X -0.336,Y -488.086,Z 259.544,A 0.000,B 0.000,C 90.000,E1 134.028} C_DIS
LIN {X 0.128,Y -488.126,Z 259.539,A 0.000,B 0.000,C 90.000,E1 133.056} C_DIS
LIN {X -0.071,Y -487.876,Z 259.534,A 0.000,B 0.000,C 90.000,E1 132.162} C_DIS
LIN {X 0.059,Y -487.384,Z 259.529,A 0.000,B 0.000,C 90.000,E1 131.229} C_DIS
LIN {X -0.138,Y -486.650,Z 259.524,A 0.000,B 0.000,C 90.000,E1 130.334} C_DIS
LIN {X 0.303,Y -485.122,Z 259.516,A 0.000,B 0.000,C 90.000,E1 128.749} C_DIS
LIN {X -0.103,Y -483.748,Z 259.509,A 0.000,B 0.000,C 90.000,E1 127.569} C_DIS
LIN {X 0.238,Y -482.059,Z 259.502,A 0.000,B 0.000,C 90.000,E1 126.297} C_DIS
LIN {X 0.074,Y -480.655,Z 259.497,A 0.000,B 0.000,C 90.000,E1 125.391} C_DIS
LIN {X -0.296,Y -477.564,Z 259.486,A 0.000,B 0.000,C 90.000,E1 123.579} C_DIS
LIN {X 0.056,Y -474.314,Z 259.476,A 0.000,B 0.000,C 90.000,E1 121.671} C_DIS
LIN {X -0.098,Y -471.487,Z 259.467,A 0.000,B 0.000,C 90.000,E1 120.129} C_DIS
LIN {X -0.129,Y -468.643,Z 259.459,A 0.000,B 0.000,C 90.000,E1 118.565} C_DIS
LIN {X -0.071,Y -465.266,Z 259.448,A 0.000,B 0.000,C 90.000,E1 116.668} C_DIS
LIN {X -0.097,Y -461.768,Z 259.438,A 0.000,B 0.000,C 90.000,E1 114.771} C_DIS
LIN {X 0.119,Y -458.949,Z 259.429,A 0.000,B 0.000,C 90.000,E1 113.153} C_DIS
LIN {X 0.094,Y -455.094,Z 259.416,A 0.000,B 0.000,C 90.000,E1 110.918} C_DIS
LIN {X -0.140,Y -454.732,Z 259.415,A 0.000,B 0.000,C 90.000,E1 110.737} C_DIS
LIN {X -0.180,Y -454.743,Z 259.415,A 0.000,B 0.000,C 90.000,E1 110.737} C_DIS
LIN {X 0.221,Y -456.818,Z 259.411,A 0.000,B 0.000,C 90.000,E1 109.939} C_DIS
LIN {X 0.124,Y -457.564,Z 259.409,A 0.000,B 0.000,C 90.000,E1 109.631} C_DIS
LIN {X 0.211,Y -466.263,Z 259.386,A 0.000,B 0.000,C 90.000,E1 105.481} C_DIS
LIN {X -0.187,Y -467.818,Z 259.383,A 0.000,B 0.000,C 90.000,E1 104.898} C_DIS
LIN {X -0.216,Y -476.025,Z 259.357,A 0.000,B 0.000,C 90.000,E1 100.197} C_DIS
LIN {X 0.088,Y -477.352,Z 259.350,A 0.000,B 0.000,C 90.000,E1 98.916} C_DIS
LIN {X 0.057,Y -481.958,Z 259.331,A 0.000,B 0.000,C 90.000,E1 95.511} C_DIS
LIN {X 0.190,Y -482.349,Z 259.327,A 0.000,B 0.000,C 90.000,E1 94.878} C_DIS
LIN {X -0.157,Y -485.420,Z 259.305,A 0.000,B 0.000,C 90.000,E1 90.917} C_DIS
LIN {X 0.153,Y -485.527,Z 259.303,A 0.000,B 0.000,C 90.000,E1 90.573} C_DIS
LIN {X -0.125,Y -486.372,Z 259.281,A 0.000,B 0.000,C 90.000,E1 86.617} C_DIS
LIN {X 0.186,Y -486.366,Z 259.279,A 0.000,B 0.000,C 90.000,E1 86.274} C_DIS
LIN {X 0.199,Y -485.362,Z 259.269,A 0.000,B 0.000,C 90.000,E1 84.432} C_DIS
LIN {X 0.203,Y -484.691,Z 259.254,A 0.000,B 0.000,C 90.000,E1 81.667} C_DIS
LIN {X 0.071,Y -484.472,Z 259.252,A 0.000,B 0.000,C 90.000,E1 81.376} C_DIS
LIN {X 0.075,Y -480.655,Z 259.228,A 0.000,B 0.000,C 90.000,E1 77.061} C_DIS
LIN {X 0.041,Y -480.393,Z 259.227,A 0.000,B 0.000,C 90.000,E1 76.756} C_DIS
LIN {X -0.186,Y -474.180,Z 259.201,A 0.000,B 0.000,C 90.000,E1 72.127} C_DIS
LIN {X 0.162,Y -472.372,Z 259.195,A 0.000,B 0.000,C 90.000,E1 71.148} C_DIS
LIN {X 0.073,Y -467.947,Z 259.181,A 0.000,B 0.000,C 90.000,E1 68.646} C_DIS
LIN {X 0.033,Y -467.951,Z 259.181,A 0.000,B 0.000,C 90.000,E1 68.646} C_DIS
LIN {X -0.203,Y -473.586,Z 259.169,A 0.000,B 0.000,C 90.000,E1 66.485} C_DIS
LIN {X 0.015,Y -478.468,Z 259.159,A 0.000,B 0.000,C 90.000,E1 64.588} C_DIS
LIN {X 0.128,Y -484.241,Z 259.147,A 0.000,B 0.000,C 90.000,E1 62.410} C_DIS
LIN {X -0.051,Y -489.296,Z 259.137,A 0.000,B 0.000,C 90.000,E1 60.589} C_DIS
LIN {X 0.119,Y -494.561,Z 259.126,A 0.000,B 0.000,C 90.000,E1 58.742} C_DIS
LIN {X -0.044,Y -498.863,Z 259.118,A 0.000,B 0.000,C 90.000,E1 57.248} C_DIS
LIN {X 0.272,Y -502.178,Z 259.111,A 0.000,B 0.000,C 90.000,E1 56.008} C_DIS
LIN {X -0.175,Y -506.122,Z 259.103,A 0.000,B 0.000,C 90.000,E1 54.562} C_DIS
LIN {X 0.130,Y -509.108,Z 259.096,A 0.000,B 0.000,C 90.000,E1 53.336} C_DIS
LIN {X -0.316,Y -512.487,Z 259.088,A 0.000,B 0.000,C 90.000,E1 51.904} C_DIS
LIN {X 0.085,Y -514.939,Z 259.082,A 0.000,B 0.000,C 90.000,E1 50.678} C_DIS
LIN {X -0.277,Y -517.134,Z 259.075,A 0.000,B 0.000,C 90.000,E1 49.542} C_DIS
LIN {X 0.193,Y -518.525,Z 259.070,A 0.000,B 0.000,C 90.000,E1 48.609} C_DIS
LIN {X -0.047,Y -519.793,Z 259.065,A 0.000,B 0.000,C 90.000,E1 47.757} C_DIS
LIN {X 0.017,Y -521.185,Z 259.059,A 0.000,B 0.000,C 90.000,E1 46.581} C_DIS
LIN {X -0.200,Y -521.993,Z 259.054,A 0.000,B 0.000,C 90.000,E1 45.729} C_DIS
LIN {X -0.045,Y -522.624,Z 259.049,A 0.000,B 0.000,C 90.000,E1 44.838} C_DIS
LIN {X 0.055,Y -523.157,Z 259.043,A 0.000,B 0.000,C 90.000,E1 43.662} C_DIS
LIN {X -0.218,Y -523.447,Z 259.036,A 0.000,B 0.000,C 90.000,E1 42.528} C_DIS
LIN {X -0.018,Y -523.538,Z 259.031,A 0.000,B 0.000,C 90.000,E1 41.634} C_DIS
LIN {X -0.206,Y -523.477,Z 259.026,A 0.000,B 0.000,C 90.000,E1 40.782} C_DIS
LIN {X 0.000,Y -523.215,Z 259.022,A 0.000,B 0.000,C 90.000,E1 39.886} C_DIS
LIN {X -0.246,Y -522.580,Z 259.015,A 0.000,B 0.000,C 90.000,E1 38.749} C_DIS
LIN {X -0.103,Y -521.805,Z 259.009,A 0.000,B 0.000,C 90.000,E1 37.569} C_DIS
LIN {X 0.125,Y -520.744,Z 259.002,A 0.000,B 0.000,C 90.000,E1 36.377} C_DIS
LIN {X -0.025,Y -519.748,Z 258.997,A 0.000,B 0.000,C 90.000,E1 35.518} C_DIS
LIN {X -0.236,Y -517.521,Z 258.988,A 0.000,B 0.000,C 90.000,E1 33.785} C_DIS
LIN {X -0.075,Y -515.910,Z 258.981,A 0.000,B 0.000,C 90.000,E1 32.594} C_DIS
LIN {X 0.215,Y -513.485,Z 258.971,A 0.000,B 0.000,C 90.000,E1 30.797} C_DIS
LIN {X -0.242,Y -511.228,Z 258.961,A 0.000,B 0.000,C 90.000,E1 29.077} C_DIS
LIN {X 0.145,Y -509.014,Z 258.952,A 0.000,B 0.000,C 90.000,E1 27.257} C_DIS
LIN {X 0.246,Y -506.872,Z 258.942,A 0.000,B 0.000,C 90.000,E1 25.463} C_DIS
LIN {X 0.078,Y -505.003,Z 258.932,A 0.000,B 0.000,C 90.000,E1 23.695} C_DIS
LIN {X 0.046,Y -503.467,Z 258.923,A 0.000,B 0.000,C 90.000,E1 22.206} C_DIS
LIN {X -0.196,Y -502.062,Z 258.915,A 0.000,B 0.000,C 90.000,E1 20.737} C_DIS
LIN {X 0.151,Y -500.260,Z 258.903,A 0.000,B 0.000,C 90.000,E1 18.598} C_DIS
LIN {X 0.035,Y -498.306,Z 258.890,A 0.000,B 0.000,C 90.000,E1 16.205} C_DIS
LIN {X 0.214,Y -496.622,Z 258.877,A 0.000,B 0.000,C 90.000,E1 13.772} C_DIS
LIN {X 0.200,Y -495.472,Z 258.865,A 0.000,B 0.000,C 90.000,E1 11.658} C_DIS
LIN {X -0.133,Y -494.412,Z 258.850,A 0.000,B 0.000,C 90.000,E1 8.973} C_DIS
LIN {X 0.019,Y -493.997,Z 258.838,A 0.000,B 0.000,C 90.000,E1 6.834} C_DIS
LIN {X 0.173,Y -493.905,Z 258.821,A 0.000,B 0.000,C 90.000,E1 3.784} C_DIS
LIN {X 0.174,Y -494.228,Z 258.809,A 0.000,B 0.000,C 90.000,E1 1.661} C_DIS
LIN {X -0.023,Y -495.745,Z 258.790,A 0.000,B 0.000,C 90.000,E1 358.282} C_DIS
LIN {X -0.209,Y -497.761,Z 258.775,A 0.000,B 0.000,C 90.000,E1 355.584} C_DIS
LIN {X 0.114,Y -503.328,Z 258.749,A 0.000,B 0.000,C 90.000,E1 350.735} C_DIS
LIN {X 0.258,Y -506.622,Z 258.739,A 0.000,B 0.000,C 90.000,E1 348.926} C_DIS
LIN {X -0.091,Y -515.600,Z 258.719,A 0.000,B 0.000,C 90.000,E1 345.408} C_DIS
LIN {X 0.207,Y -520.333,Z 258.709,A 0.000,B 0.000,C 90.000,E1 343.614} C_DIS
LIN {X -0.049,Y -528.517,Z 258.693,A 0.000,B 0.000,C 90.000,E1 340.732} C_DIS
LIN {X -0.187,Y -536.871,Z 258.679,A 0.000,B 0.000,C 90.000,E1 338.156} C_DIS
LIN {X -0.297,Y -541.734,Z 258.671,A 0.000,B 0.000,C 90.000,E1 336.741} C_DIS
LIN {X 0.115,Y -546.647,Z 258.663,A 0.000,B 0.000,C 90.000,E1 335.281} C_DIS
LIN {X -0.073,Y -553.736,Z 258.652,A 0.000,B 0.000,C 90.000,E1 333.332} C_DIS
LIN {X 0.116,Y -560.019,Z 258.643,A 0.000,B 0.000,C 90.000,E1 331.641} C_DIS
LIN {X 0.065,Y -564.164,Z 258.636,A 0.000,B 0.000,C 90.000,E1 330.539} C_DIS
LIN {X -0.140,Y -568.141,Z 258.630,A 0.000,B 0.000,C 90.000,E1 329.459} C_DIS
LIN {X 0.028,Y -572.932,Z 258.623,A 0.000,B 0.000,C 90.000,E1 328.074} C_DIS
LIN {X 0.239,Y -580.913,Z 258.611,A 0.000,B 0.000,C 90.000,E1 325.881} C_DIS
LIN {X -0.039,Y -586.084,Z 258.603,A 0.000,B 0.000,C 90.000,E1 324.562} C_DIS
LIN {X -0.091,Y -590.011,Z 258.597,A 0.000,B 0.000,C 90.000,E1 323.497} C_DIS
LIN {X -0.346,Y -594.555,Z 258.590,A 0.000,B 0.000,C 90.000,E1 322.190} C_DIS
LIN {X 0.328,Y -600.709,Z 258.580,A 0.000,B 0.000,C 90.000,E1 320.275} C_DIS
LIN {X -0.214,Y -605.163,Z 258.572,A 0.000,B 0.000,C 90.000,E1 319.013} C_DIS
LIN {X 0.200,Y -611.429,Z 258.562,A 0.000,B 0.000,C 90.000,E1 317.148} C_DIS
LIN {X 0.117,Y -614.170,Z 258.558,A 0.000,B 0.000,C 90.000,E1 316.377} C_DIS
LIN {X 0.056,Y -616.696,Z 258.553,A 0.000,B 0.000,C 90.000,E1 315.607} C_DIS
LIN {X -0.140,Y -619.803,Z 258.548,A 0.000,B 0.000,C 90.000,E1 314.595} C_DIS
LIN {X 0.145,Y -622.563,Z 258.542,A 0.000,B 0.000,C 90.000,E1 313.542} C_DIS
LIN {X 0.038,Y -625.156,Z 258.536,A 0.000,B 0.000,C 90.000,E1 312.528} C_DIS
LIN {X 0.095,Y -626.944,Z 258.532,A 0.000,B 0.000,C 90.000,E1 311.757} C_DIS
LIN {X 0.171,Y -628.527,Z 258.528,A 0.000,B 0.000,C 90.000,E1 310.987} C_DIS
LIN {X -0.148,Y -630.007,Z 258.524,A 0.000,B 0.000,C 90.000,E1 310.253} C_DIS
LIN {X -0.047,Y -631.378,Z 258.519,A 0.000,B 0.000,C 90.000,E1 309.483} C_DIS
LIN {X 0.031,Y -632.873,Z 258.514,A 0.000,B 0.000,C 90.000,E1 308.463} C_DIS
LIN {X 0.132,Y -634.195,Z 258.508,A 0.000,B 0.000,C 90.000,E1 307.443} C_DIS
LIN {X -0.133,Y -635.241,Z 258.503,A 0.000,B 0.000,C 90.000,E1 306.457} C_DIS
LIN {X 0.125,Y -635.772,Z 258.498,A 0.000,B 0.000,C 90.000,E1 305.678} C_DIS
LIN {X -0.134,Y -636.041,Z 258.494,A 0.000,B 0.000,C 90.000,E1 304.945} C_DIS
LIN {X 0.172,Y -636.221,Z 258.487,A 0.000,B 0.000,C 90.000,E1 303.658} C_DIS
LIN {X 0.082,Y -636.076,Z 258.483,A 0.000,B 0.000,C 90.000,E1 302.911} C_DIS
LIN {X 0.331,Y -635.639,Z 258.479,A 0.000,B 0.000,C 90.000,E1 302.133} C_DIS
LIN {X -0.102,Y -634.869,Z 258.475,A 0.000,B 0.000,C 90.000,E1 301.416} C_DIS
LIN {X -0.208,Y -633.838,Z 258.470,A 0.000,B 0.000,C 90.000,E1 300.669} C_DIS
LIN {X -0.298,Y -631.998,Z 258.465,A 0.000,B 0.000,C 90.000,E1 299.667} C_DIS
LIN {X 0.132,Y -629.860,Z 258.459,A 0.000,B 0.000,C 90.000,E1 298.615} C_DIS
LIN {X -0.301,Y -626.830,Z 258.452,A 0.000,B 0.000,C 90.000,E1 297.385} C_DIS
LIN {X -0.235,Y -624.153,Z 258.446,A 0.000,B 0.000,C 90.000,E1 296.360} C_DIS
LIN {X -0.208,Y -621.400,Z 258.441,A 0.000,B 0.000,C 90.000,E1 295.335} C_DIS
LIN {X -0.239,Y -615.275,Z 258.428,A 0.000,B 0.000,C 90.000,E1 293.025} C_DIS
LIN {X -0.365,Y -610.705,Z 258.418,A 0.000,B 0.000,C 90.000,E1 291.227} C_DIS
LIN {X -0.251,Y -606.407,Z 258.408,A 0.000,B 0.000,C 90.000,E1 289.396} C_DIS
LIN {X -0.237,Y -601.179,Z 258.395,A 0.000,B 0.000,C 90.000,E1 287.040} C_DIS
LIN {X 0.134,Y -598.019,Z 258.386,A 0.000,B 0.000,C 90.000,E1 285.426} C_DIS
LIN {X 0.247,Y -593.377,Z 258.371,A 0.000,B 0.000,C 90.000,E1 282.771} C_DIS
LIN {X -0.039,Y -589.724,Z 258.356,A 0.000,B 0.000,C 90.000,E1 280.141} C_DIS
LIN {X 0.021,Y -586.216,Z 258.337,A 0.000,B 0.000,C 90.000,E1 276.663} C_DIS
LIN {X -0.274,Y -584.571,Z 258.322,A 0.000,B 0.000,C 90.000,E1 274.012} C_DIS
LIN {X 0.234,Y -583.868,Z 258.309,A 0.000,B 0.000,C 90.000,E1 271.547} C_DIS
LIN {X -0.153,Y -585.009,Z 258.283,A 0.000,B 0.000,C 90.000,E1 267.020} C_DIS
LIN {X 0.093,Y -587.875,Z 258.264,A 0.000,B 0.000,C 90.000,E1 263.514} C_DIS
LIN {X 0.125,Y -590.381,Z 258.252,A 0.000,B 0.000,C 90.000,E1 261.376} C_DIS
LIN {X -0.299,Y -594.252,Z 258.237,A 0.000,B 0.000,C 90.000,E1 258.757} C_DIS
LIN {X -0.060,Y -597.120,Z 258.227,A 0.000,B 0.000,C 90.000,E1 256.881} C_DIS
LIN {X -0.062,Y -598.742,Z 258.221,A 0.000,B 0.000,C 90.000,E1 255.825} C_DIS
LIN {X -0.191,Y -599.985,Z 258.217,A 0.000,B 0.000,C 90.000,E1 255.046} C_DIS
LIN {X -0.001,Y -601.417,Z 258.211,A 0.000,B 0.000,C 90.000,E1 253.976} C_DIS
LIN {X -0.092,Y -602.387,Z 258.207,A 0.000,B 0.000,C 90.000,E1 253.196} C_DIS
LIN {X -0.173,Y -603.056,Z 258.202,A 0.000,B 0.000,C 90.000,E1 252.417} C_DIS
LIN {X 0.044,Y -603.632,Z 258.196,A 0.000,B 0.000,C 90.000,E1 251.348} C_DIS
LIN {X 0.085,Y -603.908,Z 258.191,A 0.000,B 0.000,C 90.000,E1 250.296} C_DIS
LIN {X -0.066,Y -603.967,Z 258.185,A 0.000,B 0.000,C 90.000,E1 249.263} C_DIS
LIN {X 0.067,Y -603.612,Z 258.180,A 0.000,B 0.000,C 90.000,E1 248.465} C_DIS
LIN {X 0.193,Y -603.022,Z 258.176,A 0.000,B 0.000,C 90.000,E1 247.667} C_DIS
LIN {X -0.245,Y -602.227,Z 258.172,A 0.000,B 0.000,C 90.000,E1 246.922} C_DIS
LIN {X 0.101,Y -601.254,Z 258.167,A 0.000,B 0.000,C 90.000,E1 246.102} C_DIS
LIN {X 0.188,Y -599.935,Z 258.163,A 0.000,B 0.000,C 90.000,E1 245.305} C_DIS
LIN {X -0.035,Y -598.391,Z 258.159,A 0.000,B 0.000,C 90.000,E1 244.537} C_DIS
LIN {X 0.183,Y -596.063,Z 258.153,A 0.000,B 0.000,C 90.000,E1 243.461} C_DIS
LIN {X 0.014,Y -592.833,Z 258.145,A 0.000,B 0.000,C 90.000,E1 242.153} C_DIS
LIN {X -0.094,Y -590.078,Z 258.139,A 0.000,B 0.000,C 90.000,E1 241.101} C_DIS
LIN {X 0.273,Y -587.179,Z 258.134,A 0.000,B 0.000,C 90.000,E1 239.999} C_DIS
LIN {X 0.079,Y -584.027,Z 258.128,A 0.000,B 0.000,C 90.000,E1 238.948} C_DIS
LIN {X 0.284,Y -581.512,Z 258.123,A 0.000,B 0.000,C 90.000,E1 238.122} C_DIS
LIN {X 0.155,Y -577.137,Z 258.116,A 0.000,B 0.000,C 90.000,E1 236.786} C_DIS
LIN {X 0.060,Y -571.031,Z 258.105,A 0.000,B 0.000,C 90.000,E1 234.895} C_DIS
LIN {X 0.043,Y -565.968,Z 258.096,A 0.000,B 0.000,C 90.000,E1 233.256} C_DIS
LIN {X 0.014,Y -560.031,Z 258.085,A 0.000,B 0.000,C 90.000,E1 231.331} C_DIS
LIN {X 0.369,Y -555.797,Z 258.078,A 0.000,B 0.000,C 90.000,E1 229.908} C_DIS
LIN {X 0.287,Y -550.631,Z 258.068,A 0.000,B 0.000,C 90.000,E1 228.243} C_DIS
LIN {X 0.054,Y -546.200,Z 258.060,A 0.000,B 0.000,C 90.000,E1 226.863} C_DIS
LIN {X 0.108,Y -540.792,Z 258.051,A 0.000,B 0.000,C 90.000,E1 225.162} C_DIS
LIN {X -0.312,Y -536.273,Z 258.043,A 0.000,B 0.000,C 90.000,E1 223.785} C_DIS
LIN {X -0.088,Y -530.918,Z 258.034,A 0.000,B 0.000,C 90.000,E1 222.043} C_DIS
LIN {X 0.050,Y -525.581,Z 258.024,A 0.000,B 0.000,C 90.000,E1 220.297} C_DIS
LIN {X 0.141,Y -520.373,Z 258.014,A 0.000,B 0.000,C 90.000,E1 218.543} C_DIS
LIN {X 0.185,Y -516.071,Z 258.006,A 0.000,B 0.000,C 90.000,E1 217.076} C_DIS
LIN {X 0.170,Y -511.058,Z 257.996,A 0.000,B 0.000,C 90.000,E1 215.311} C_DIS
LIN {X 0.078,Y -505.166,Z 257.985,A 0.000,B 0.000,C 90.000,E1 213.245} C_DIS
LIN {X 0.256,Y -499.526,Z 257.973,A 0.000,B 0.000,C 90.000,E1 211.131} C_DIS
LIN {X -0.105,Y -495.697,Z 257.965,A 0.000,B 0.000,C 90.000,E1 209.667} C_DIS
LIN {X 0.002,Y -489.130,Z 257.950,A 0.000,B 0.000,C 90.000,E1 206.924} C_DIS
LIN {X 0.114,Y -483.286,Z 257.934,A 0.000,B 0.000,C 90.000,E1 204.155} C_DIS
LIN {X -0.154,Y -477.878,Z 257.919,A 0.000,B 0.000,C 90.000,E1 201.408} C_DIS
LIN {X -0.038,Y -473.564,Z 257.905,A 0.000,B 0.000,C 90.000,E1 198.906} C_DIS
LIN {X -0.116,Y -470.677,Z 257.895,A 0.000,B 0.000,C 90.000,E1 197.040} C_DIS
LIN {X 0.061,Y -466.687,Z 257.879,A 0.000,B 0.000,C 90.000,E1 194.189} C_DIS
LIN {X 0.081,Y -463.541,Z 257.865,A 0.000,B 0.000,C 90.000,E1 191.658} C_DIS
LIN {X 0.025,Y -460.895,Z 257.853,A 0.000,B 0.000,C 90.000,E1 189.443} C_DIS
LIN {X -0.227,Y -458.017,Z 257.837,A 0.000,B 0.000,C 90.000,E1 186.606} C_DIS
LIN {X 0.109,Y -456.306,Z 257.826,A 0.000,B 0.000,C 90.000,E1 184.645} C_DIS
LIN {X -0.232,Y -454.309,Z 257.812,A 0.000,B 0.000,C 90.000,E1 182.121} C_DIS
LIN {X 0.093,Y -452.810,Z 257.799,A 0.000,B 0.000,C 90.000,E1 179.828} C_DIS
LIN {X 0.090,Y -451.495,Z 257.785,A 0.000,B 0.000,C 90.000,E1 177.249} C_DIS
LIN {X 0.087,Y -450.710,Z 257.770,A 0.000,B 0.000,C 90.000,E1 174.666} C_DIS
LIN {X 0.061,Y -450.514,Z 257.762,A 0.000,B 0.000,C 90.000,E1 173.053} C_DIS
LIN {X 0.038,Y -450.551,Z 257.749,A 0.000,B 0.000,C 90.000,E1 170.792} C_DIS
LIN {X 0.097,Y -450.848,Z 257.736,A 0.000,B 0.000,C 90.000,E1 168.522} C_DIS
LIN {X 0.050,Y -451.466,Z 257.726,A 0.000,B 0.000,C 90.000,E1 166.589} C_DIS
LIN {X -0.016,Y -452.250,Z 257.713,A 0.000,B 0.000,C 90.000,E1 164.338} C_DIS
LIN {X -0.054,Y -454.591,Z 257.692,A 0.000,B 0.000,C 90.000,E1 160.477} C_DIS
LIN {X -0.159,Y -456.690,Z 257.677,A 0.000,B 0.000,C 90.000,E1 157.922} C_DIS
LIN {X -0.024,Y -458.994,Z 257.665,A 0.000,B 0.000,C 90.000,E1 155.665} C_DIS
LIN {X -0.158,Y -461.244,Z 257.654,A 0.000,B 0.000,C 90.000,E1 153.768} C_DIS
LIN {X -0.264,Y -465.088,Z 257.638,A 0.000,B 0.000,C 90.000,E1 150.923} C_DIS
LIN {X 0.138,Y -468.400,Z 257.626,A 0.000,B 0.000,C 90.000,E1 148.663} C_DIS
LIN {X -0.004,Y -472.487,Z 257.612,A 0.000,B 0.000,C 90.000,E1 146.167} C_DIS
LIN {X -0.045,Y -475.117,Z 257.603,A 0.000,B 0.000,C 90.000,E1 144.609} C_DIS
LIN {X -0.230,Y -478.081,Z 257.593,A 0.000,B 0.000,C 90.000,E1 142.763} C_DIS
LIN {X 0.130,Y -480.421,Z 257.584,A 0.000,B 0.000,C 90.000,E1 141.170} C_DIS
LIN {X 0.154,Y -482.545,Z 257.576,A 0.000,B 0.000,C 90.000,E1 139.622} C_DIS
LIN {X 0.218,Y -483.709,Z 257.571,A 0.000,B 0.000,C 90.000,E1 138.690} C_DIS
LIN {X 0.114,Y -484.978,Z 257.564,A 0.000,B 0.000,C 90.000,E1 137.472} C_DIS
LIN {X 0.207,Y -485.742,Z 257.559,A 0.000,B 0.000,C 90.000,E1 136.539} C_DIS
LIN {X -0.041,Y -486.292,Z 257.554,A 0.000,B 0.000,C 90.000,E1 135.648} C_DIS
LIN {X 0.061,Y -486.639,Z 257.549,A 0.000,B 0.000,C 90.000,E1 134.717} C_DIS
LIN {X 0.170,Y -486.850,Z 257.543,A 0.000,B 0.000,C 90.000,E1 133.785} C_DIS
LIN {X -0.253,Y -486.801,Z 257.537,A 0.000,B 0.000,C 90.000,E1 132.609} C_DIS
LIN {X -0.137,Y -486.425,Z 257.531,A 0.000,B 0.000,C 90.000,E1 131.676} C_DIS
LIN {X -0.029,Y -485.794,Z 257.526,A 0.000,B 0.000,C 90.000,E1 130.744} C_DIS
LIN {X 0.080,Y -484.376,Z 257.518,A 0.000,B 0.000,C 90.000,E1 129.197} C_DIS
LIN {X 0.047,Y -483.095,Z 257.511,A 0.000,B 0.000,C 90.000,E1 127.971} C_DIS
LIN {X -0.202,Y -481.952,Z 257.506,A 0.000,B 0.000,C 90.000,E1 127.076} C_DIS
LIN {X 0.115,Y -480.224,Z 257.499,A 0.000,B 0.000,C 90.000,E1 125.804} C_DIS
LIN {X -0.067,Y -477.700,Z 257.490,A 0.000,B 0.000,C 90.000,E1 124.278} C_DIS
LIN {X -0.086,Y -475.633,Z 257.484,A 0.000,B 0.000,C 90.000,E1 123.038} C_DIS
LIN {X 0.041,Y -472.891,Z 257.475,A 0.000,B 0.000,C 90.000,E1 121.465} C_DIS
LIN {X -0.141,Y -470.080,Z 257.466,A 0.000,B 0.000,C 90.000,E1 119.922} C_DIS
LIN {X -0.201,Y -467.251,Z 257.457,A 0.000,B 0.000,C 90.000,E1 118.359} C_DIS
LIN {X 0.028,Y -463.905,Z 257.447,A 0.000,B 0.000,C 90.000,E1 116.437} C_DIS
LIN {X 0.174,Y -460.393,Z 257.436,A 0.000,B 0.000,C 90.000,E1 114.515} C_DIS
LIN {X -0.061,Y -457.594,Z 257.428,A 0.000,B 0.000,C 90.000,E1 112.950} C_DIS
LIN {X 0.099,Y -454.171,Z 257.416,A 0.000,B 0.000,C 90.000,E1 110.918} C_DIS
LIN {X 0.059,Y -454.175,Z 257.416,A 0.000,B 0.000,C 90.000,E1 110.918} C_DIS
LIN {X -0.172,Y -457.404,Z 257.410,A 0.000,B 0.000,C 90.000,E1 109.758} C_DIS
LIN {X -0.089,Y -466.046,Z 257.387,A 0.000,B 0.000,C 90.000,E1 105.607} C_DIS
LIN {X 0.085,Y -467.615,Z 257.383,A 0.000,B 0.000,C 90.000,E1 104.954} C_DIS
LIN {X 0.083,Y -469.069,Z 257.378,A 0.000,B 0.000,C 90.000,E1 104.008} C_DIS
LIN {X 0.044,Y -475.839,Z 257.357,A 0.000,B 0.000,C 90.000,E1 100.254} C_DIS
LIN {X -0.118,Y -476.322,Z 257.355,A 0.000,B 0.000,C 90.000,E1 99.962} C_DIS
LIN {X -0.172,Y -481.818,Z 257.331,A 0.000,B 0.000,C 90.000,E1 95.625} C_DIS
LIN {X 0.156,Y -482.178,Z 257.329,A 0.000,B 0.000,C 90.000,E1 95.277} C_DIS
LIN {X 0.090,Y -485.327,Z 257.306,A 0.000,B 0.000,C 90.000,E1 90.974} C_DIS
LIN {X -0.086,Y -485.535,Z 257.304,A 0.000,B 0.000,C 90.000,E1 90.688} C_DIS
LIN {X 0.122,Y -486.328,Z 257.282,A 0.000,B 0.000,C 90.000,E1 86.674} C_DIS
LIN {X -0.229,Y -486.292,Z 257.278,A 0.000,B 0.000,C 90.000,E1 86.102} C_DIS
LIN {X -0.024,Y -484.695,Z 257.254,A 0.000,B 0.000,C 90.000,E1 81.781} C_DIS
LIN {X -0.156,Y -484.578,Z 257.253,A 0.000,B 0.000,C 90.000,E1 81.489} C_DIS
LIN {X 0.193,Y -480.516,Z 257.227,A 0.000,B 0.000,C 90.000,E1 76.825} C_DIS
LIN {X 0.088,Y -474.267,Z 257.201,A 0.000,B 0.000,C 90.000,E1 72.181} C_DIS
LIN {X 0.056,Y -473.810,Z 257.199,A 0.000,B 0.000,C 90.000,E1 71.873} C_DIS
LIN {X 0.059,Y -467.583,Z 257.180,A 0.000,B 0.000,C 90.000,E1 68.411} C_DIS
LIN {X 0.019,Y -467.585,Z 257.180,A 0.000,B 0.000,C 90.000,E1 68.411} C_DIS
LIN {X 0.032,Y -473.219,Z 257.168,A 0.000,B 0.000,C 90.000,E1 66.230} C_DIS
LIN {X 0.040,Y -478.065,Z 257.158,A 0.000,B 0.000,C 90.000,E1 64.357} C_DIS
LIN {X 0.140,Y -483.009,Z 257.147,A 0.000,B 0.000,C 90.000,E1 62.487} C_DIS
LIN {X 0.164,Y -488.911,Z 257.135,A 0.000,B 0.000,C 90.000,E1 60.333} C_DIS
LIN {X 0.062,Y -493.295,Z 257.127,A 0.000,B 0.000,C 90.000,E1 58.820} C_DIS
LIN {X -0.128,Y -497.605,Z 257.118,A 0.000,B 0.000,C 90.000,E1 57.327} C_DIS
LIN {X 0.163,Y -500.879,Z 257.112,A 0.000,B 0.000,C 90.000,E1 56.087} C_DIS
LIN {X 0.094,Y -504.086,Z 257.105,A 0.000,B 0.000,C 90.000,E1 54.895} C_DIS
LIN {X -0.029,Y -507.828,Z 257.097,A 0.000,B 0.000,C 90.000,E1 53.417} C_DIS
LIN {X 0.217,Y -511.176,Z 257.089,A 0.000,B 0.000,C 90.000,E1 51.904} C_DIS
LIN {X 0.201,Y -513.646,Z 257.082,A 0.000,B 0.000,C 90.000,E1 50.723} C_DIS
LIN {X 0.297,Y -515.311,Z 257.077,A 0.000,B 0.000,C 90.000,E1 49.828} C_DIS
LIN {X 0.020,Y -516.849,Z 257.072,A 0.000,B 0.000,C 90.000,E1 48.976} C_DIS
LIN {X 0.077,Y -518.480,Z 257.066,A 0.000,B 0.000,C 90.000,E1 47.796} C_DIS
LIN {X 0.184,Y -519.533,Z 257.061,A 0.000,B 0.000,C 90.000,E1 46.905} C_DIS
LIN {X -0.049,Y -520.404,Z 257.056,A 0.000,B 0.000,C 90.000,E1 46.053} C_DIS
LIN {X 0.088,Y -521.094,Z 257.051,A 0.000,B 0.000,C 90.000,E1 45.162} C_DIS
LIN {X 0.233,Y -521.593,Z 257.046,A 0.000,B 0.000,C 90.000,E1 44.271} C_DIS
LIN {X 0.022,Y -521.928,Z 257.041,A 0.000,B 0.000,C 90.000,E1 43.419} C_DIS
LIN {X 0.115,Y -522.190,Z 257.035,A 0.000,B 0.000,C 90.000,E1 42.243} C_DIS
LIN {X 0.205,Y -522.258,Z 257.028,A 0.000,B 0.000,C 90.000,E1 41.067} C_DIS
LIN {X -0.054,Y -521.906,Z 257.022,A 0.000,B 0.000,C 90.000,E1 39.930} C_DIS
LIN {X 0.130,Y -521.450,Z 257.017,A 0.000,B 0.000,C 90.000,E1 39.036} C_DIS
LIN {X -0.065,Y -520.687,Z 257.010,A 0.000,B 0.000,C 90.000,E1 37.890} C_DIS
LIN {X 0.048,Y -519.698,Z 257.004,A 0.000,B 0.000,C 90.000,E1 36.710} C_DIS
LIN {X 0.303,Y -518.731,Z 256.999,A 0.000,B 0.000,C 90.000,E1 35.804} C_DIS
LIN {X -0.229,Y -517.217,Z 256.993,A 0.000,B 0.000,C 90.000,E1 34.692} C_DIS
LIN {X -0.137,Y -515.255,Z 256.984,A 0.000,B 0.000,C 90.000,E1 33.214} C_DIS
LIN {X 0.139,Y -512.779,Z 256.975,A 0.000,B 0.000,C 90.000,E1 31.416} C_DIS
LIN {X -0.093,Y -509.637,Z 256.962,A 0.000,B 0.000,C 90.000,E1 29.077} C_DIS
LIN {X 0.256,Y -507.398,Z 256.952,A 0.000,B 0.000,C 90.000,E1 27.257} C_DIS
LIN {X -0.135,Y -505.226,Z 256.942,A 0.000,B 0.000,C 90.000,E1 25.515} C_DIS
LIN {X 0.117,Y -503.357,Z 256.932,A 0.000,B 0.000,C 90.000,E1 23.695} C_DIS
LIN {X -0.024,Y -502.146,Z 256.925,A 0.000,B 0.000,C 90.000,E1 22.514} C_DIS
LIN {X -0.111,Y -500.732,Z 256.917,A 0.000,B 0.000,C 90.000,E1 21.025} C_DIS
LIN {X -0.039,Y -499.134,Z 256.907,A 0.000,B 0.000,C 90.000,E1 19.214} C_DIS
LIN {X 0.105,Y -497.830,Z 256.898,A 0.000,B 0.000,C 90.000,E1 17.692} C_DIS
LIN {X -0.033,Y -496.425,Z 256.888,A 0.000,B 0.000,C 90.000,E1 15.898} C_DIS
LIN {X 0.051,Y -494.974,Z 256.877,A 0.000,B 0.000,C 90.000,E1 13.772} C_DIS
LIN {X -0.005,Y -493.824,Z 256.865,A 0.000,B 0.000,C 90.000,E1 11.658} C_DIS
LIN {X 0.195,Y -492.821,Z 256.851,A 0.000,B 0.000,C 90.000,E1 9.208} C_DIS
LIN {X -0.177,Y -492.350,Z 256.840,A 0.000,B 0.000,C 90.000,E1 7.125} C_DIS
LIN {X 0.030,Y -492.120,Z 256.829,A 0.000,B 0.000,C 90.000,E1 5.277} C_DIS
LIN {X 0.142,Y -492.206,Z 256.819,A 0.000,B 0.000,C 90.000,E1 3.440} C_DIS
LIN {X -0.047,Y -492.700,Z 256.806,A 0.000,B 0.000,C 90.000,E1 1.031} C_DIS
LIN {X -0.187,Y -494.164,Z 256.789,A 0.000,B 0.000,C 90.000,E1 357.993} C_DIS
LIN {X 0.192,Y -495.981,Z 256.775,A 0.000,B 0.000,C 90.000,E1 355.527} C_DIS
LIN {X -0.016,Y -501.052,Z 256.750,A 0.000,B 0.000,C 90.000,E1 351.027} C_DIS
LIN {X 0.073,Y -504.204,Z 256.740,A 0.000,B 0.000,C 90.000,E1 349.218} C_DIS
LIN {X 0.186,Y -511.464,Z 256.724,A 0.000,B 0.000,C 90.000,E1 346.228} C_DIS
LIN {X 0.150,Y -515.472,Z 256.715,A 0.000,B 0.000,C 90.000,E1 344.755} C_DIS
LIN {X -0.183,Y -519.439,Z 256.707,A 0.000,B 0.000,C 90.000,E1 343.323} C_DIS
LIN {X -0.143,Y -528.644,Z 256.689,A 0.000,B 0.000,C 90.000,E1 340.115} C_DIS
LIN {X -0.187,Y -535.278,Z 256.678,A 0.000,B 0.000,C 90.000,E1 338.103} C_DIS
LIN {X 0.107,Y -541.126,Z 256.669,A 0.000,B 0.000,C 90.000,E1 336.357} C_DIS
LIN {X -0.209,Y -546.068,Z 256.661,A 0.000,B 0.000,C 90.000,E1 334.973} C_DIS
LIN {X 0.035,Y -550.084,Z 256.655,A 0.000,B 0.000,C 90.000,E1 333.819} C_DIS
LIN {X -0.100,Y -556.366,Z 256.645,A 0.000,B 0.000,C 90.000,E1 332.153} C_DIS
LIN {X -0.201,Y -560.595,Z 256.639,A 0.000,B 0.000,C 90.000,E1 331.051} C_DIS
LIN {X 0.034,Y -564.634,Z 256.633,A 0.000,B 0.000,C 90.000,E1 329.921} C_DIS
LIN {X 0.146,Y -569.506,Z 256.625,A 0.000,B 0.000,C 90.000,E1 328.535} C_DIS
LIN {X -0.053,Y -577.416,Z 256.613,A 0.000,B 0.000,C 90.000,E1 326.373} C_DIS
LIN {X -0.222,Y -583.694,Z 256.604,A 0.000,B 0.000,C 90.000,E1 324.769} C_DIS
LIN {X -0.308,Y -587.635,Z 256.598,A 0.000,B 0.000,C 90.000,E1 323.703} C_DIS
LIN {X 0.019,Y -591.321,Z 256.592,A 0.000,B 0.000,C 90.000,E1 322.603} C_DIS
LIN {X 0.261,Y -595.711,Z 256.585,A 0.000,B 0.000,C 90.000,E1 321.251} C_DIS
LIN {X -0.345,Y -602.002,Z 256.575,A 0.000,B 0.000,C 90.000,E1 319.461} C_DIS
LIN {X -0.025,Y -606.529,Z 256.567,A 0.000,B 0.000,C 90.000,E1 318.119} C_DIS
LIN {X -0.030,Y -612.939,Z 256.557,A 0.000,B 0.000,C 90.000,E1 316.296} C_DIS
LIN {X 0.327,Y -615.510,Z 256.553,A 0.000,B 0.000,C 90.000,E1 315.486} C_DIS
LIN {X -0.316,Y -618.639,Z 256.547,A 0.000,B 0.000,C 90.000,E1 314.514} C_DIS
LIN {X -0.049,Y -621.384,Z 256.541,A 0.000,B 0.000,C 90.000,E1 313.461} C_DIS
LIN {X -0.173,Y -623.909,Z 256.536,A 0.000,B 0.000,C 90.000,E1 312.447} C_DIS
LIN {X -0.130,Y -625.694,Z 256.532,A 0.000,B 0.000,C 90.000,E1 311.676} C_DIS
LIN {X 0.272,Y -627.712,Z 256.526,A 0.000,B 0.000,C 90.000,E1 310.620} C_DIS
LIN {X -0.183,Y -629.603,Z 256.520,A 0.000,B 0.000,C 90.000,E1 309.644} C_DIS
LIN {X -0.128,Y -631.088,Z 256.515,A 0.000,B 0.000,C 90.000,E1 308.624} C_DIS
LIN {X -0.028,Y -632.097,Z 256.510,A 0.000,B 0.000,C 90.000,E1 307.855} C_DIS
LIN {X 0.190,Y -632.979,Z 256.506,A 0.000,B 0.000,C 90.000,E1 307.076} C_DIS
LIN {X -0.090,Y -633.663,Z 256.502,A 0.000,B 0.000,C 90.000,E1 306.343} C_DIS
LIN {X -0.226,Y -634.133,Z 256.498,A 0.000,B 0.000,C 90.000,E1 305.598} C_DIS
LIN {X 0.017,Y -634.351,Z 256.493,A 0.000,B 0.000,C 90.000,E1 304.818} C_DIS
LIN {X 0.276,Y -634.533,Z 256.488,A 0.000,B 0.000,C 90.000,E1 303.785} C_DIS
LIN {X 0.168,Y -634.418,Z 256.484,A 0.000,B 0.000,C 90.000,E1 303.038} C_DIS
LIN {X 0.060,Y -634.009,Z 256.479,A 0.000,B 0.000,C 90.000,E1 302.291} C_DIS
LIN {X -0.052,Y -633.292,Z 256.475,A 0.000,B 0.000,C 90.000,E1 301.544} C_DIS
LIN {X -0.175,Y -632.319,Z 256.471,A 0.000,B 0.000,C 90.000,E1 300.797} C_DIS
LIN {X 0.233,Y -631.031,Z 256.467,A 0.000,B 0.000,C 90.000,E1 300.001} C_DIS
LIN {X 0.100,Y -629.014,Z 256.461,A 0.000,B 0.000,C 90.000,E1 298.999} C_DIS
LIN {X 0.145,Y -627.905,Z 256.458,A 0.000,B 0.000,C 90.000,E1 298.487} C_DIS
LIN {X -0.318,Y -624.842,Z 256.451,A 0.000,B 0.000,C 90.000,E1 297.257} C_DIS
LIN {X -0.275,Y -621.433,Z 256.444,A 0.000,B 0.000,C 90.000,E1 295.976} C_DIS
LIN {X 0.281,Y -619.365,Z 256.440,A 0.000,B 0.000,C 90.000,E1 295.155} C_DIS
LIN {X 0.161,Y -612.622,Z 256.426,A 0.000,B 0.000,C 90.000,E1 292.589} C_DIS
LIN {X 0.203,Y -606.871,Z 256.413,A 0.000,B 0.000,C 90.000,E1 290.248} C_DIS
LIN {X -0.270,Y -603.265,Z 256.404,A 0.000,B 0.000,C 90.000,E1 288.725} C_DIS
LIN {X -0.078,Y -597.698,Z 256.389,A 0.000,B 0.000,C 90.000,E1 286.079} C_DIS
LIN {X -0.140,Y -592.422,Z 256.373,A 0.000,B 0.000,C 90.000,E1 283.175} C_DIS
LIN {X -0.211,Y -588.279,Z 256.357,A 0.000,B 0.000,C 90.000,E1 280.254} C_DIS
LIN {X -0.116,Y -585.879,Z 256.345,A 0.000,B 0.000,C 90.000,E1 278.106} C_DIS
LIN {X -0.225,Y -584.761,Z 256.338,A 0.000,B 0.000,C 90.000,E1 276.777} C_DIS
LIN {X -0.035,Y -583.082,Z 256.323,A 0.000,B 0.000,C 90.000,E1 274.073} C_DIS
LIN {X -0.279,Y -582.498,Z 256.296,A 0.000,B 0.000,C 90.000,E1 269.255} C_DIS
LIN {X -0.036,Y -583.951,Z 256.279,A 0.000,B 0.000,C 90.000,E1 266.274} C_DIS
LIN {X 0.165,Y -586.334,Z 256.264,A 0.000,B 0.000,C 90.000,E1 263.571} C_DIS
LIN {X -0.170,Y -589.196,Z 256.251,A 0.000,B 0.000,C 90.000,E1 261.197} C_DIS
LIN {X 0.268,Y -592.724,Z 256.238,A 0.000,B 0.000,C 90.000,E1 258.757} C_DIS
LIN {X -0.109,Y -595.557,Z 256.227,A 0.000,B 0.000,C 90.000,E1 256.937} C_DIS
LIN {X 0.163,Y -596.784,Z 256.223,A 0.000,B 0.000,C 90.000,E1 256.117} C_DIS
LIN {X 0.306,Y -598.444,Z 256.217,A 0.000,B 0.000,C 90.000,E1 255.046} C_DIS
LIN {X -0.102,Y -599.863,Z 256.211,A 0.000,B 0.000,C 90.000,E1 254.031} C_DIS
LIN {X -0.095,Y -600.581,Z 256.208,A 0.000,B 0.000,C 90.000,E1 253.504} C_DIS
LIN {X -0.198,Y -601.320,Z 256.204,A 0.000,B 0.000,C 90.000,E1 252.725} C_DIS
LIN {X 0.183,Y -602.022,Z 256.198,A 0.000,B 0.000,C 90.000,E1 251.638} C_DIS
LIN {X 0.005,Y -602.344,Z 256.192,A 0.000,B 0.000,C 90.000,E1 250.604} C_DIS
LIN {X -0.167,Y -602.473,Z 256.186,A 0.000,B 0.000,C 90.000,E1 249.571} C_DIS
LIN {X 0.026,Y -602.406,Z 256.184,A 0.000,B 0.000,C 90.000,E1 249.028} C_DIS
LIN {X -0.126,Y -602.165,Z 256.181,A 0.000,B 0.000,C 90.000,E1 248.518} C_DIS
LIN {X -0.313,Y -601.309,Z 256.175,A 0.000,B 0.000,C 90.000,E1 247.486} C_DIS
LIN {X 0.019,Y -600.465,Z 256.170,A 0.000,B 0.000,C 90.000,E1 246.666} C_DIS
LIN {X 0.103,Y -599.400,Z 256.166,A 0.000,B 0.000,C 90.000,E1 245.869} C_DIS
LIN {X -0.127,Y -598.034,Z 256.162,A 0.000,B 0.000,C 90.000,E1 245.101} C_DIS
LIN {X 0.006,Y -595.251,Z 256.154,A 0.000,B 0.000,C 90.000,E1 243.768} C_DIS
LIN {X 0.178,Y -592.719,Z 256.148,A 0.000,B 0.000,C 90.000,E1 242.692} C_DIS
LIN {X -0.047,Y -589.423,Z 256.141,A 0.000,B 0.000,C 90.000,E1 241.385} C_DIS
LIN {X -0.205,Y -586.520,Z 256.135,A 0.000,B 0.000,C 90.000,E1 240.333} C_DIS
LIN {X -0.107,Y -583.417,Z 256.129,A 0.000,B 0.000,C 90.000,E1 239.253} C_DIS
LIN {X -0.207,Y -580.932,Z 256.125,A 0.000,B 0.000,C 90.000,E1 238.456} C_DIS
LIN {X -0.025,Y -576.588,Z 256.117,A 0.000,B 0.000,C 90.000,E1 237.089} C_DIS
LIN {X -0.035,Y -568.693,Z 256.104,A 0.000,B 0.000,C 90.000,E1 234.642} C_DIS
LIN {X 0.115,Y -564.475,Z 256.096,A 0.000,B 0.000,C 90.000,E1 233.256} C_DIS
LIN {X 0.048,Y -558.508,Z 256.085,A 0.000,B 0.000,C 90.000,E1 231.331} C_DIS
LIN {X -0.054,Y -555.118,Z 256.079,A 0.000,B 0.000,C 90.000,E1 230.231} C_DIS
LIN {X -0.154,Y -549.953,Z 256.070,A 0.000,B 0.000,C 90.000,E1 228.566} C_DIS
LIN {X -0.026,Y -545.536,Z 256.062,A 0.000,B 0.000,C 90.000,E1 227.148} C_DIS
LIN {X 0.028,Y -540.124,Z 256.053,A 0.000,B 0.000,C 90.000,E1 225.445} C_DIS
LIN {X -0.026,Y -535.604,Z 256.045,A 0.000,B 0.000,C 90.000,E1 224.028} C_DIS
LIN {X 0.159,Y -529.330,Z 256.033,A 0.000,B 0.000,C 90.000,E1 222.000} C_DIS
LIN {X -0.129,Y -523.967,Z 256.024,A 0.000,B 0.000,C 90.000,E1 220.297} C_DIS
LIN {X -0.073,Y -518.765,Z 256.014,A 0.000,B 0.000,C 90.000,E1 218.543} C_DIS
